KUKA KRL program: MyProgram_077().src

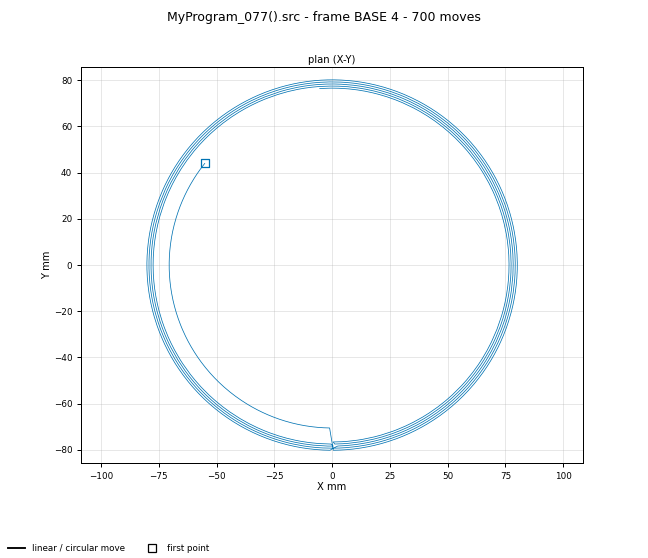
[picture p0: tool path of MyProgram_077().src in frame BASE 4, 700 of 700 moves have a stored position in this frame; points joined in program order, loops and branches not executed]
&ACCESS RVP
&REL 1
&PARAM TEMPLATE = C:\KRC\Roboter\Template\vorgabe
&PARAM EDITMASK = *
DEF MyProgram_077()
; ---- Setting reference (Base) ----
$BASE = BASE_DATA[4]

; --------------------------
; ---- Setting tool (TCP) ----
$TOOL = TOOL_DATA[3]
; --------------------------

$VEL.CP = VEL_APROX_PRINT
Startdeposition()
$VEL.CP = VEL_PRINT
LIN {X -55.1314,Y 43.9885,Z 79,A 136.1081,B 24.8816,C -2.5111,E1 24.8737,E2 308.1338} C_DIS
LIN {X -57.0335,Y 41.4919,Z 79,A 138.4284,B 24.8828,C -2.4992,E1 24.8699,E2 305.8307} C_DIS
LIN {X -58.5164,Y 39.3729,Z 79,A 140.5439,B 24.8833,C -2.4938,E1 24.8665,E2 303.7176} C_DIS
LIN {X -59.694,Y 37.5637,Z 79,A 142.4917,B 24.8833,C -2.4932,E1 24.8636,E2 301.7614} C_DIS
LIN {X -61.332,Y 34.8263,Z 79,A 145.2364,B 24.8837,C -2.4892,E1 24.8597,E2 299.012} C_DIS
LIN {X -62.6132,Y 32.4671,Z 79,A 147.3566,B 24.8844,C -2.4816,E1 24.857,E2 296.8988} C_DIS
LIN {X -63.7621,Y 30.1485,Z 79,A 149.3257,B 24.8853,C -2.4725,E1 24.8546,E2 294.9408} C_DIS
LIN {X -64.8254,Y 27.7886,Z 79,A 151.5952,B 24.8855,C -2.4698,E1 24.8521,E2 292.665} C_DIS
LIN {X -65.8013,Y 25.3913,Z 79,A 153.5568,B 24.8864,C -2.4604,E1 24.8501,E2 290.715} C_DIS
LIN {X -66.6884,Y 22.9605,Z 79,A 155.8268,B 24.8866,C -2.4576,E1 24.8479,E2 288.4387} C_DIS
LIN {X -67.5472,Y 20.2926,Z 79,A 158.0661,B 24.8874,C -2.4498,E1 24.8461,E2 286.2053} C_DIS
LIN {X -68.3657,Y 17.3357,Z 79,A 160.5177,B 24.8882,C -2.4412,E1 24.8443,E2 283.76} C_DIS
LIN {X -69.0025,Y 14.601,Z 79,A 162.777,B 24.8889,C -2.4335,E1 24.843,E2 281.5058} C_DIS
LIN {X -69.4922,Y 12.0572,Z 79,A 165.0492,B 24.8891,C -2.4305,E1 24.8418,E2 279.2273} C_DIS
LIN {X -69.9406,Y 9.0919,Z 79,A 167.3407,B 24.8901,C -2.4197,E1 24.8409,E2 276.948} C_DIS
LIN {X -70.2503,Y 6.2684,Z 79,A 169.5832,B 24.8909,C -2.4109,E1 24.8403,E2 274.7129} C_DIS
LIN {X -70.4338,Y 3.6722,Z 79,A 171.7072,B 24.8915,C -2.4044,E1 24.8399,E2 272.5917} C_DIS
LIN {X -70.5211,Y 1.0827,Z 79,A 174.0196,B 24.8917,C -2.4023,E1 24.8398,E2 270.2705} C_DIS
LIN {X -70.5092,Y -1.7264,Z 79,A 176.375,B 24.8922,C -2.3966,E1 24.8398,E2 267.9144} C_DIS
LIN {X -70.3982,Y -4.3149,Z 79,A 178.3488,B 24.8931,C -2.3871,E1 24.8402,E2 265.9514} C_DIS
LIN {X -70.1904,Y -6.9165,Z 79,A -179.3706,B 24.8934,C -2.384,E1 24.8408,E2 263.6647} C_DIS
LIN {X -69.8585,Y -9.7054,Z 79,A -177.1426,B 24.8941,C -2.3757,E1 24.8416,E2 261.4432} C_DIS
LIN {X -69.455,Y -12.2641,Z 79,A -175.0214,B 24.8946,C -2.3696,E1 24.8425,E2 259.324} C_DIS
LIN {X -68.8624,Y -15.2436,Z 79,A -172.5842,B 24.8954,C -2.3613,E1 24.8439,E2 256.8921} C_DIS
LIN {X -68.2017,Y -17.9741,Z 79,A -170.1696,B 24.8957,C -2.3573,E1 24.8456,E2 254.473} C_DIS
LIN {X -67.4309,Y -20.6756,Z 79,A -167.9357,B 24.8964,C -2.3495,E1 24.8474,E2 252.2449} C_DIS
LIN {X -66.6291,Y -23.1294,Z 79,A -165.8252,B 24.8969,C -2.3436,E1 24.8492,E2 250.1363} C_DIS
LIN {X -65.5843,Y -25.9438,Z 79,A -163.5524,B 24.8979,C -2.3329,E1 24.8515,E2 247.8763} C_DIS
LIN {X -64.775,Y -27.9042,Z 79,A -161.562,B 24.8978,C -2.334,E1 24.8537,E2 245.8724} C_DIS
LIN {X -63.4784,Y -30.7391,Z 79,A -159.2749,B 24.8989,C -2.3215,E1 24.8564,E2 243.6027} C_DIS
LIN {X -62.3075,Y -33.0479,Z 79,A -157.1577,B 24.8994,C -2.3161,E1 24.8591,E2 241.4871} C_DIS
LIN {X -61.053,Y -35.3117,Z 79,A -154.9151,B 24.8996,C -2.3136,E1 24.8622,E2 239.2385} C_DIS
LIN {X -59.5877,Y -37.7339,Z 79,A -152.4789,B 24.8998,C -2.3108,E1 24.8658,E2 236.7968} C_DIS
LIN {X -58.1586,Y -39.9012,Z 79,A -150.364,B 24.9003,C -2.3056,E1 24.8691,E2 234.6836} C_DIS
LIN {X -56.6707,Y -41.9875,Z 79,A -148.288,B 24.9007,C -2.3004,E1 24.8725,E2 232.61} C_DIS
LIN {X -54.7949,Y -44.4057,Z 79,A -145.763,B 24.9011,C -2.2955,E1 24.8769,E2 230.0849} C_DIS
LIN {X -52.7706,Y -46.7945,Z 79,A -143.2185,B 24.9016,C -2.2898,E1 24.8815,E2 227.5425} C_DIS
LIN {X -50.8754,Y -48.8473,Z 79,A -141.0304,B 24.9022,C -2.283,E1 24.8857,E2 225.3609} C_DIS
LIN {X -48.8605,Y -50.8627,Z 79,A -138.5931,B 24.9024,C -2.2811,E1 24.8906,E2 222.9182} C_DIS
LIN {X -46.6368,Y -52.9099,Z 79,A -136.1496,B 24.9028,C -2.276,E1 24.8956,E2 220.4769} C_DIS
LIN {X -44.1609,Y -54.9933,Z 79,A -133.5445,B 24.9033,C -2.2706,E1 24.9013,E2 217.8749} C_DIS
LIN {X -41.7925,Y -56.8134,Z 79,A -131.1597,B 24.9037,C -2.2654,E1 24.9066,E2 215.4938} C_DIS
LIN {X -39.3679,Y -58.5198,Z 79,A -128.7599,B 24.9041,C -2.2613,E1 24.9121,E2 213.0956} C_DIS
LIN {X -37.0061,Y -60.0423,Z 79,A -126.3522,B 24.9041,C -2.2608,E1 24.9178,E2 210.6814} C_DIS
LIN {X -34.7597,Y -61.3701,Z 79,A -124.3781,B 24.9047,C -2.2544,E1 24.9225,E2 208.7168} C_DIS
LIN {X -32.4884,Y -62.6022,Z 79,A -122.1216,B 24.9046,C -2.2555,E1 24.9281,E2 206.4514} C_DIS
LIN {X -30.1741,Y -63.7499,Z 79,A -120.1783,B 24.9051,C -2.2493,E1 24.933,E2 204.5179} C_DIS
LIN {X -27.8222,Y -64.8108,Z 79,A -117.9214,B 24.9049,C -2.2509,E1 24.9388,E2 202.2517} C_DIS
LIN {X -25.4477,Y -65.7792,Z 79,A -115.9713,B 24.9054,C -2.2457,E1 24.9438,E2 200.3098} C_DIS
LIN {X -22.9341,Y -66.6975,Z 79,A -113.6524,B 24.9052,C -2.2474,E1 24.95,E2 197.9823} C_DIS
LIN {X -20.263,Y -67.556,Z 79,A -111.4377,B 24.9055,C -2.2442,E1 24.9558,E2 195.7714} C_DIS
LIN {X -17.3572,Y -68.3602,Z 79,A -109.033,B 24.9057,C -2.2416,E1 24.9623,E2 193.3691} C_DIS
LIN {X -14.6256,Y -68.9972,Z 79,A -106.7919,B 24.9059,C -2.2396,E1 24.9684,E2 191.13} C_DIS
LIN {X -12.087,Y -69.4868,Z 79,A -104.5246,B 24.9056,C -2.2431,E1 24.9747,E2 188.8521} C_DIS
LIN {X -9.24,Y -69.9214,Z 79,A -102.2807,B 24.9059,C -2.2402,E1 24.9809,E2 186.6133} C_DIS
LIN {X -6.2929,Y -70.248,Z 79,A -100.0258,B 24.9062,C -2.2361,E1 24.9871,E2 184.3669} C_DIS
LIN {X -3.7214,Y -70.431,Z 79,A -97.9292,B 24.9062,C -2.2361,E1 24.993,E2 182.2693} C_DIS
LIN {X -1.0857,Y -70.521,Z 79,A -95.6624,B 24.9059,C -2.2397,E1 24.9993,E2 179.994} C_DIS
LIN {X -1.0857,Y -70.521,Z 79,A -95.6624,B 24.9059,C -2.2397,E1 24.9993,E2 179.994} C_DIS
Enddeposition()
LIN {X 0.5223,Y -80.1629,Z 80,A -94.9522,B 24.9201,C -2.0638,E1 25.0001,E2 179.7014} C_DIS
Startdeposition()
$VEL.CP = VEL_PRINT
LIN {X 3.5738,Y -80.0857,Z 80,A -91.9127,B 24.9181,C -2.0895,E1 25.0088,E2 176.6013} C_DIS
LIN {X 6.2912,Y -79.9181,Z 80,A -90.0185,B 24.9181,C -2.0889,E1 25.0141,E2 174.7096} C_DIS
LIN {X 9.0357,Y -79.6549,Z 80,A -87.8669,B 24.9177,C -2.0954,E1 25.0201,E2 172.544} C_DIS
LIN {X 12.4392,Y -79.1945,Z 80,A -85.4934,B 24.9177,C -2.0946,E1 25.0266,E2 170.1743} C_DIS
LIN {X 15.6125,Y -78.6306,Z 80,A -83.3311,B 24.9179,C -2.0923,E1 25.0325,E2 168.0202} C_DIS
LIN {X 18.3183,Y -78.0448,Z 80,A -81.1674,B 24.9173,C -2.0997,E1 25.0385,E2 165.8418} C_DIS
LIN {X 21.381,Y -77.2609,Z 80,A -79.2279,B 24.9179,C -2.0924,E1 25.0437,E2 163.9226} C_DIS
LIN {X 24.237,Y -76.415,Z 80,A -76.7008,B 24.9168,C -2.1069,E1 25.0505,E2 161.3657} C_DIS
LIN {X 27.8769,Y -75.1616,Z 80,A -74.34,B 24.9174,C -2.0985,E1 25.0566,E2 159.0296} C_DIS
LIN {X 30.4325,Y -74.1645,Z 80,A -72.076,B 24.9165,C -2.1105,E1 25.0626,E2 156.7422} C_DIS
LIN {X 33.383,Y -72.8834,Z 80,A -70.0419,B 24.9168,C -2.1058,E1 25.0677,E2 154.7241} C_DIS
LIN {X 36.0435,Y -71.606,Z 80,A -67.7149,B 24.916,C -2.1159,E1 25.0736,E2 152.3794} C_DIS
LIN {X 38.7509,Y -70.1782,Z 80,A -65.5829,B 24.9159,C -2.1179,E1 25.0788,E2 150.2488} C_DIS
LIN {X 41.2637,Y -68.7311,Z 80,A -63.4611,B 24.9155,C -2.1232,E1 25.0839,E2 148.121} C_DIS
LIN {X 43.8675,Y -67.0985,Z 80,A -61.3015,B 24.9152,C -2.1263,E1 25.089,E2 145.9611} C_DIS
LIN {X 46.5483,Y -65.2666,Z 80,A -59.038,B 24.915,C -2.1292,E1 25.0942,E2 143.6986} C_DIS
LIN {X 49.1868,Y -63.3027,Z 80,A -56.5823,B 24.9143,C -2.1374,E1 25.0997,E2 141.2324} C_DIS
LIN {X 51.8574,Y -61.1335,Z 80,A -54.1898,B 24.914,C -2.1408,E1 25.1048,E2 138.8411} C_DIS
LIN {X 54.4427,Y -58.8436,Z 80,A -51.7288,B 24.9136,C -2.1462,E1 25.1099,E2 136.3771} C_DIS
LIN {X 56.7655,Y -56.6064,Z 80,A -49.4236,B 24.9132,C -2.1518,E1 25.1145,E2 134.0685} C_DIS
LIN {X 58.9533,Y -54.3231,Z 80,A -47.1689,B 24.9127,C -2.1572,E1 25.1188,E2 131.8108} C_DIS
LIN {X 61.3516,Y -51.6011,Z 80,A -44.5862,B 24.9122,C -2.1635,E1 25.1235,E2 129.2249} C_DIS
LIN {X 63.3027,Y -49.1868,Z 80,A -42.3804,B 24.9118,C -2.1689,E1 25.1274,E2 127.0165} C_DIS
LIN {X 65.2666,Y -46.5483,Z 80,A -40.0511,B 24.9113,C -2.1746,E1 25.1312,E2 124.6851} C_DIS
LIN {X 67.0985,Y -43.8675,Z 80,A -37.7702,B 24.9109,C -2.1798,E1 25.1347,E2 122.4033} C_DIS
LIN {X 68.7749,Y -41.19,Z 80,A -35.5455,B 24.9104,C -2.1851,E1 25.138,E2 120.1774} C_DIS
LIN {X 70.2553,Y -38.6115,Z 80,A -33.4541,B 24.91,C -2.1902,E1 25.1408,E2 118.0849} C_DIS
LIN {X 71.6694,Y -35.9177,Z 80,A -31.2202,B 24.9093,C -2.1985,E1 25.1437,E2 115.8433} C_DIS
LIN {X 72.9727,Y -33.1892,Z 80,A -29.1799,B 24.9091,C -2.201,E1 25.1461,E2 113.8079} C_DIS
LIN {X 74.1645,Y -30.4325,Z 80,A -26.9676,B 24.9084,C -2.2096,E1 25.1485,E2 111.5875} C_DIS
LIN {X 75.3506,Y -27.3635,Z 80,A -24.62,B 24.9078,C -2.2167,E1 25.1508,E2 109.2362} C_DIS
LIN {X 76.4315,Y -24.1845,Z 80,A -22.1399,B 24.907,C -2.2267,E1 25.153,E2 106.7466} C_DIS
LIN {X 77.5189,Y -20.4316,Z 80,A -19.4725,B 24.9066,C -2.2314,E1 25.1549,E2 104.0834} C_DIS
LIN {X 78.2582,Y -17.3842,Z 80,A -17.344,B 24.9063,C -2.2348,E1 25.1563,E2 101.9592} C_DIS
LIN {X 78.8279,Y -14.5873,Z 80,A -15.2763,B 24.9057,C -2.2422,E1 25.1574,E2 99.8862} C_DIS
LIN {X 79.2987,Y -11.7628,Z 80,A -13.2188,B 24.9051,C -2.2491,E1 25.1583,E2 97.8246} C_DIS
LIN {X 79.6766,Y -8.836,Z 80,A -11.0985,B 24.9045,C -2.2562,E1 25.159,E2 95.7} C_DIS
LIN {X 79.9651,Y -5.6668,Z 80,A -8.7996,B 24.9038,C -2.2642,E1 25.1595,E2 93.3958} C_DIS
LIN {X 80.1418,Y -1.9398,Z 80,A -6.211,B 24.9033,C -2.2702,E1 25.1598,E2 90.8084} C_DIS
LIN {X 80.1574,Y 1.1669,Z 80,A -3.8994,B 24.9025,C -2.2802,E1 25.1598,E2 88.487} C_DIS
LIN {X 80.0402,Y 4.4763,Z 80,A -1.6758,B 24.9022,C -2.2831,E1 25.1594,E2 86.2697} C_DIS
LIN {X 79.8147,Y 7.4897,Z 80,A 0.4758,B 24.9016,C -2.2896,E1 25.1589,E2 84.1155} C_DIS
LIN {X 79.4367,Y 10.7888,Z 80,A 2.902,B 24.9009,C -2.2988,E1 25.1581,E2 81.682} C_DIS
LIN {X 78.9428,Y 13.9486,Z 80,A 5.1167,B 24.9004,C -2.3036,E1 25.1571,E2 79.4689} C_DIS
LIN {X 78.398,Y 16.7433,Z 80,A 7.168,B 24.8999,C -2.3104,E1 25.1559,E2 77.4136} C_DIS
LIN {X 77.6572,Y 19.8955,Z 80,A 9.4494,B 24.8993,C -2.3164,E1 25.1544,E2 75.1312} C_DIS
LIN {X 76.9876,Y 22.3515,Z 80,A 11.3758,B 24.8986,C -2.3252,E1 25.1529,E2 73.1948} C_DIS
LIN {X 75.804,Y 26.0855,Z 80,A 14.1035,B 24.898,C -2.3312,E1 25.1505,E2 70.4684} C_DIS
LIN {X 74.7866,Y 28.8732,Z 80,A 16.2095,B 24.8975,C -2.3369,E1 25.1484,E2 68.3608} C_DIS
LIN {X 73.5077,Y 31.9859,Z 80,A 18.5391,B 24.8971,C -2.3414,E1 25.1459,E2 66.0335} C_DIS
LIN {X 72.4161,Y 34.3876,Z 80,A 20.5035,B 24.8965,C -2.3491,E1 25.1436,E2 64.0613} C_DIS
LIN {X 70.8869,Y 37.437,Z 80,A 22.7713,B 24.8963,C -2.3504,E1 25.1407,E2 61.8024} C_DIS
LIN {X 69.5058,Y 39.9426,Z 80,A 24.807,B 24.8959,C -2.3556,E1 25.1379,E2 59.7651} C_DIS
LIN {X 67.9275,Y 42.5716,Z 80,A 27.0111,B 24.8953,C -2.3617,E1 25.1347,E2 57.5578} C_DIS
LIN {X 66.2424,Y 45.1494,Z 80,A 29.2856,B 24.8946,C -2.3696,E1 25.1311,E2 55.276} C_DIS
LIN {X 64.3571,Y 47.7997,Z 80,A 31.6145,B 24.8941,C -2.3754,E1 25.1273,E2 52.9446} C_DIS
LIN {X 62.2366,Y 50.528,Z 80,A 34.0403,B 24.8937,C -2.3799,E1 25.1231,E2 50.5195} C_DIS
LIN {X 60.0369,Y 53.1237,Z 80,A 36.4824,B 24.8932,C -2.3857,E1 25.1186,E2 48.0746} C_DIS
LIN {X 57.7753,Y 55.5742,Z 80,A 38.7345,B 24.8931,C -2.3868,E1 25.1143,E2 45.8297} C_DIS
LIN {X 55.4573,Y 57.8879,Z 80,A 41.1215,B 24.8925,C -2.3931,E1 25.1095,E2 43.4378} C_DIS
LIN {X 53.0243,Y 60.1252,Z 80,A 43.5607,B 24.8919,C -2.4002,E1 25.1045,E2 40.9917} C_DIS
LIN {X 50.4022,Y 62.3385,Z 80,A 45.8875,B 24.8919,C -2.4009,E1 25.0995,E2 38.672} C_DIS
LIN {X 47.7997,Y 64.3571,Z 80,A 48.2922,B 24.8913,C -2.4066,E1 25.0941,E2 36.2627} C_DIS
LIN {X 45.1494,Y 66.2424,Z 80,A 50.5578,B 24.8911,C -2.4086,E1 25.0889,E2 33.9999} C_DIS
LIN {X 42.5716,Y 67.9275,Z 80,A 52.7489,B 24.8908,C -2.4117,E1 25.0838,E2 31.8086} C_DIS
LIN {X 39.9426,Y 69.5058,Z 80,A 54.8968,B 24.8907,C -2.4136,E1 25.0786,E2 29.6629} C_DIS
LIN {X 37.437,Y 70.8869,Z 80,A 57.0166,B 24.8902,C -2.4186,E1 25.0734,E2 27.5373} C_DIS
LIN {X 34.3002,Y 72.4573,Z 80,A 59.5962,B 24.8897,C -2.4238,E1 25.0669,E2 24.9523} C_DIS
LIN {X 31.0661,Y 73.9011,Z 80,A 62.0481,B 24.8897,C -2.4241,E1 25.0606,E2 22.5054} C_DIS
LIN {X 28.2922,Y 75.0069,Z 80,A 64.1764,B 24.8895,C -2.426,E1 25.0551,E2 20.3772} C_DIS
LIN {X 25.5016,Y 76.001,Z 80,A 66.2855,B 24.8895,C -2.4276,E1 25.0495,E2 18.2686} C_DIS
LIN {X 22.3279,Y 76.9943,Z 80,A 68.7742,B 24.8889,C -2.4326,E1 25.0428,E2 15.7724} C_DIS
LIN {X 18.9606,Y 77.8907,Z 80,A 71.1195,B 24.8892,C -2.4298,E1 25.0365,E2 13.4372} C_DIS
LIN {X 16.0165,Y 78.5487,Z 80,A 73.323,B 24.889,C -2.4322,E1 25.0305,E2 11.2309} C_DIS
LIN {X 12.7079,Y 79.153,Z 80,A 75.6013,B 24.8892,C -2.4294,E1 25.0242,E2 8.9617} C_DIS
LIN {X 9.9558,Y 79.5454,Z 80,A 77.6865,B 24.8889,C -2.4327,E1 25.0184,E2 6.8704} C_DIS
LIN {X 6.8781,Y 79.8707,Z 80,A 79.89,B 24.8889,C -2.4327,E1 25.0123,E2 4.6683} C_DIS
LIN {X 3.8564,Y 80.0735,Z 80,A 82.0431,B 24.8889,C -2.4323,E1 25.0063,E2 2.5169} C_DIS
LIN {X 0.8877,Y 80.1613,Z 80,A 84.1718,B 24.8889,C -2.4322,E1 25.0004,E2 0.3887} C_DIS
LIN {X -1.9949,Y 80.1403,Z 80,A 86.2199,B 24.8891,C -2.4314,E1 24.9947,E2 -1.6575} C_DIS
LIN {X -4.9158,Y 80.0145,Z 80,A 88.2536,B 24.8893,C -2.429,E1 24.989,E2 -3.6862} C_DIS
LIN {X -7.4897,Y 79.8147,Z 80,A 90.1437,B 24.8893,C -2.4294,E1 24.9838,E2 -5.5782} C_DIS
LIN {X -10.7888,Y 79.4367,Z 80,A 92.5901,B 24.8892,C -2.4301,E1 24.977,E2 -8.0278} C_DIS
LIN {X -13.9486,Y 78.9428,Z 80,A 94.871,B 24.8893,C -2.4283,E1 24.9707,E2 -10.3067} C_DIS
LIN {X -16.7433,Y 78.398,Z 80,A 96.9202,B 24.8895,C -2.427,E1 24.9651,E2 -12.3552} C_DIS
LIN {X -19.8955,Y 77.6572,Z 80,A 99.1945,B 24.8898,C -2.4237,E1 24.9589,E2 -14.6248} C_DIS
LIN {X -22.3544,Y 76.9868,Z 80,A 101.1478,B 24.8896,C -2.4254,E1 24.9537,E2 -16.5853} C_DIS
LIN {X -26.0855,Y 75.804,Z 80,A 103.8912,B 24.89,C -2.4206,E1 24.9464,E2 -19.3223} C_DIS
LIN {X -28.8732,Y 74.7866,Z 80,A 106.017,B 24.8903,C -2.4179,E1 24.9409,E2 -21.4463} C_DIS
LIN {X -31.9858,Y 73.5077,Z 80,A 108.3575,B 24.8907,C -2.4128,E1 24.9349,E2 -23.7799} C_DIS
LIN {X -34.3876,Y 72.4161,Z 80,A 110.3522,B 24.8907,C -2.4128,E1 24.9298,E2 -25.7798} C_DIS
LIN {X -37.437,Y 70.8869,Z 80,A 112.6419,B 24.8915,C -2.4049,E1 24.9242,E2 -28.0567} C_DIS
LIN {X -39.9426,Y 69.5058,Z 80,A 114.6975,B 24.8918,C -2.4016,E1 24.9192,E2 -30.1106} C_DIS
LIN {X -42.5716,Y 67.9275,Z 80,A 116.9235,B 24.892,C -2.3986,E1 24.9139,E2 -32.3362} C_DIS
LIN {X -45.1494,Y 66.2424,Z 80,A 119.2205,B 24.8922,C -2.3969,E1 24.9085,E2 -34.6368} C_DIS
LIN {X -47.7997,Y 64.3571,Z 80,A 121.5729,B 24.8926,C -2.3929,E1 24.9032,E2 -36.9879} C_DIS
LIN {X -50.528,Y 62.2366,Z 80,A 124.0229,B 24.8931,C -2.3871,E1 24.8979,E2 -39.4333} C_DIS
LIN {X -53.1237,Y 60.0369,Z 80,A 126.4897,B 24.8935,C -2.3826,E1 24.8927,E2 -41.8989} C_DIS
LIN {X -55.5742,Y 57.7753,Z 80,A 128.7644,B 24.8942,C -2.3742,E1 24.8881,E2 -44.163} C_DIS
LIN {X -57.8879,Y 55.4573,Z 80,A 131.1754,B 24.8946,C -2.3704,E1 24.8833,E2 -46.5753} C_DIS
LIN {X -60.1252,Y 53.0243,Z 80,A 133.6393,B 24.8949,C -2.3672,E1 24.8787,E2 -49.0424} C_DIS
LIN {X -62.3385,Y 50.4022,Z 80,A 135.9889,B 24.8957,C -2.3582,E1 24.8746,E2 -51.3814} C_DIS
LIN {X -64.3571,Y 47.7997,Z 80,A 138.4176,B 24.896,C -2.3538,E1 24.8705,E2 -53.8114} C_DIS
LIN {X -66.2424,Y 45.1494,Z 80,A 140.7052,B 24.8967,C -2.3466,E1 24.8668,E2 -56.0929} C_DIS
LIN {X -67.9275,Y 42.5716,Z 80,A 142.931,B 24.8972,C -2.3411,E1 24.8635,E2 -58.3168} C_DIS
LIN {X -69.5058,Y 39.9426,Z 80,A 145.086,B 24.8978,C -2.3339,E1 24.8605,E2 -60.4659} C_DIS
LIN {X -70.8869,Y 37.437,Z 80,A 147.2257,B 24.8981,C -2.3304,E1 24.8576,E2 -62.6086} C_DIS
LIN {X -72.4161,Y 34.3876,Z 80,A 149.5869,B 24.8989,C -2.3213,E1 24.8547,E2 -64.9607} C_DIS
LIN {X -73.5077,Y 31.9859,Z 80,A 151.584,B 24.8991,C -2.3185,E1 24.8525,E2 -66.9621} C_DIS
LIN {X -74.7948,Y 28.8515,Z 80,A 154.0385,B 24.8997,C -2.312,E1 24.8499,E2 -69.4148} C_DIS
LIN {X -75.9027,Y 25.7931,Z 80,A 156.3282,B 24.9004,C -2.304,E1 24.8478,E2 -71.6984} C_DIS
LIN {X -76.9943,Y 22.3279,Z 80,A 159.0891,B 24.9007,C -2.3001,E1 24.8456,E2 -74.466} C_DIS
LIN {X -77.8907,Y 18.9606,Z 80,A 161.4535,B 24.9017,C -2.2891,E1 24.844,E2 -76.8179} C_DIS
LIN {X -78.5198,Y 16.1591,Z 80,A 163.4998,B 24.9023,C -2.2825,E1 24.8428,E2 -78.8604} C_DIS
LIN {X -79.0431,Y 13.3669,Z 80,A 165.555,B 24.9028,C -2.2767,E1 24.8418,E2 -80.914} C_DIS
LIN {X -79.4633,Y 10.5895,Z 80,A 167.6778,B 24.9031,C -2.2733,E1 24.841,E2 -83.0413} C_DIS
LIN {X -79.8411,Y 7.2032,Z 80,A 170.0244,B 24.9039,C -2.2632,E1 24.8403,E2 -85.378} C_DIS
LIN {X -80.0708,Y 3.9061,Z 80,A 172.4309,B 24.9044,C -2.2568,E1 24.8399,E2 -87.7836} C_DIS
LIN {X -80.1613,Y 0.8877,Z 80,A 174.553,B 24.9051,C -2.249,E1 24.8398,E2 -89.8999} C_DIS
LIN {X -80.1403,Y -1.9949,Z 80,A 176.715,B 24.9054,C -2.2451,E1 24.8398,E2 -92.0656} C_DIS
LIN {X -79.9844,Y -5.3822,Z 80,A 179.0573,B 24.9063,C -2.2354,E1 24.8402,E2 -94.3987} C_DIS
LIN {X -79.7234,Y -8.4054,Z 80,A -178.7025,B 24.9067,C -2.2304,E1 24.8408,E2 -96.6404} C_DIS
LIN {X -79.3345,Y -11.5134,Z 80,A -176.592,B 24.9075,C -2.2201,E1 24.8416,E2 -98.7389} C_DIS
LIN {X -78.9428,Y -13.9486,Z 80,A -174.6334,B 24.9075,C -2.2197,E1 24.8426,E2 -100.7082} C_DIS
LIN {X -78.398,Y -16.7433,Z 80,A -172.6016,B 24.9081,C -2.2133,E1 24.8437,E2 -102.7368} C_DIS
LIN {X -77.6572,Y -19.8955,Z 80,A -170.2891,B 24.9087,C -2.2063,E1 24.8452,E2 -105.046} C_DIS
LIN {X -76.9868,Y -22.3544,Z 80,A -168.3273,B 24.9088,C -2.2044,E1 24.8467,E2 -107.0147} C_DIS
LIN {X -75.804,Y -26.0855,Z 80,A -165.573,B 24.9096,C -2.195,E1 24.8492,E2 -109.7623} C_DIS
LIN {X -74.7866,Y -28.8732,Z 80,A -163.4397,B 24.9101,C -2.1892,E1 24.8513,E2 -111.8937} C_DIS
LIN {X -73.5077,Y -31.9858,Z 80,A -161.0918,B 24.9108,C -2.1809,E1 24.8538,E2 -114.2349} C_DIS
LIN {X -72.4161,Y -34.3876,Z 80,A -159.0914,B 24.911,C -2.1786,E1 24.8562,E2 -116.2406} C_DIS
LIN {X -70.8869,Y -37.437,Z 80,A -156.7961,B 24.9118,C -2.1682,E1 24.8591,E2 -118.5235} C_DIS
LIN {X -69.5058,Y -39.9426,Z 80,A -154.7361,B 24.9122,C -2.1632,E1 24.8619,E2 -120.5822} C_DIS
LIN {X -67.9275,Y -42.5716,Z 80,A -152.5063,B 24.9126,C -2.1585,E1 24.8652,E2 -122.8122} C_DIS
LIN {X -66.2424,Y -45.1494,Z 80,A -150.2062,B 24.9129,C -2.1555,E1 24.8687,E2 -125.1168} C_DIS
LIN {X -64.3571,Y -47.7997,Z 80,A -147.8518,B 24.9132,C -2.1506,E1 24.8726,E2 -127.4709} C_DIS
LIN {X -62.2366,Y -50.528,Z 80,A -145.4006,B 24.9138,C -2.1444,E1 24.8769,E2 -129.9187} C_DIS
LIN {X -60.0552,Y -53.1031,Z 80,A -142.9422,B 24.9141,C -2.1401,E1 24.8814,E2 -132.3782} C_DIS
LIN {X -57.7753,Y -55.5742,Z 80,A -140.6598,B 24.9148,C -2.1317,E1 24.8857,E2 -134.6504} C_DIS
LIN {X -55.4573,Y -57.8879,Z 80,A -138.2506,B 24.915,C -2.1287,E1 24.8905,E2 -137.0625} C_DIS
LIN {X -53.0243,Y -60.1252,Z 80,A -135.7897,B 24.9152,C -2.1267,E1 24.8957,E2 -139.5285} C_DIS
LIN {X -50.2555,Y -62.4575,Z 80,A -133.2988,B 24.9158,C -2.1193,E1 24.901,E2 -142.0114} C_DIS
LIN {X -47.755,Y -64.3902,Z 80,A -131.0018,B 24.916,C -2.1164,E1 24.9061,E2 -144.3096} C_DIS
LIN {X -45.1494,Y -66.2424,Z 80,A -128.7381,B 24.9163,C -2.1121,E1 24.9113,E2 -146.5709} C_DIS
LIN {X -42.5716,Y -67.9275,Z 80,A -126.5186,B 24.9166,C -2.1093,E1 24.9165,E2 -148.7907} C_DIS
LIN {X -39.9426,Y -69.5058,Z 80,A -124.3705,B 24.9169,C -2.105,E1 24.9217,E2 -150.9351} C_DIS
LIN {X -37.437,Y -70.8869,Z 80,A -122.2381,B 24.9169,C -2.1047,E1 24.9269,E2 -153.0728} C_DIS
LIN {X -34.3876,Y -72.4161,Z 80,A -119.7738,B 24.9171,C -2.1025,E1 24.9331,E2 -155.5384} C_DIS
LIN {X -31.3542,Y -73.7797,Z 80,A -117.3961,B 24.9173,C -2.1,E1 24.9392,E2 -157.9157} C_DIS
LIN {X -28.2922,Y -75.0069,Z 80,A -115.0438,B 24.9175,C -2.0977,E1 24.9453,E2 -160.2674} C_DIS
LIN {X -25.5016,Y -76.001,Z 80,A -112.9269,B 24.9176,C -2.0959,E1 24.9509,E2 -162.3843} C_DIS
LIN {X -22.3279,Y -76.9943,Z 80,A -110.4304,B 24.9175,C -2.0977,E1 24.9576,E2 -164.8891} C_DIS
LIN {X -18.9281,Y -77.8985,Z 80,A -108.0705,B 24.9179,C -2.0918,E1 24.964,E2 -167.2386} C_DIS
LIN {X -16.1591,Y -78.5198,Z 80,A -106.0453,B 24.918,C -2.0909,E1 24.9695,E2 -169.2639} C_DIS
LIN {X -13.3669,Y -79.0431,Z 80,A -104.003,B 24.918,C -2.0905,E1 24.9751,E2 -171.3075} C_DIS
LIN {X -10.5895,Y -79.4633,Z 80,A -101.8943,B 24.9178,C -2.093,E1 24.981,E2 -173.4237} C_DIS
LIN {X -7.2032,Y -79.8411,Z 80,A -99.5638,B 24.9181,C -2.0898,E1 24.9874,E2 -175.7478} C_DIS
LIN {X -3.9061,Y -80.0708,Z 80,A -97.1746,B 24.9181,C -2.0906,E1 24.9941,E2 -178.1398} C_DIS
LIN {X -0.8877,Y -80.1613,Z 80,A -95.0179,B 24.9181,C -2.0909,E1 25.0001,E2 -180.2975} C_DIS
LIN {X -0.8877,Y -80.1613,Z 80,A -95.0179,B 24.9181,C -2.0909,E1 25.0001,E2 -180.2975} C_DIS
Enddeposition()
LIN {X 0.5113,Y -79.2679,Z 80,A -94.2684,B 24.9173,C -2.0993,E1 25.0023,E2 -181.0667} C_DIS
Startdeposition()
$VEL.CP = VEL_PRINT
LIN {X -4.0138,Y -79.1697,Z 80,A -98.6051,B 24.9198,C -2.0683,E1 24.99,E2 -176.656} C_DIS
LIN {X -6.7676,Y -78.9826,Z 80,A -100.4551,B 24.9195,C -2.0724,E1 24.9849,E2 -174.8149} C_DIS
LIN {X -10.0746,Y -78.6285,Z 80,A -102.8222,B 24.9193,C -2.0738,E1 24.9783,E2 -172.4496} C_DIS
LIN {X -12.5662,Y -78.2702,Z 80,A -105.5536,B 24.9213,C -2.0491,E1 24.9706,E2 -169.6568} C_DIS
LIN {X -16.8137,Y -77.4676,Z 80,A -107.3755,B 24.9184,C -2.0864,E1 24.9659,E2 -167.9215} C_DIS
LIN {X -18.8261,Y -77.0033,Z 80,A -109.0895,B 24.9188,C -2.081,E1 24.9611,E2 -166.1924} C_DIS
LIN {X -21.2667,Y -76.3647,Z 80,A -110.994,B 24.9188,C -2.0799,E1 24.956,E2 -164.2822} C_DIS
LIN {X -24.2861,Y -75.4594,Z 80,A -113.3546,B 24.9189,C -2.0792,E1 24.9497,E2 -161.9161} C_DIS
LIN {X -27.2132,Y -74.4538,Z 80,A -115.6394,B 24.9189,C -2.0798,E1 24.9437,E2 -159.6282} C_DIS
LIN {X -30.2979,Y -73.2522,Z 80,A -118.2875,B 24.9192,C -2.0753,E1 24.9368,E2 -156.9633} C_DIS
LIN {X -33.4153,Y -71.8841,Z 80,A -121.0471,B 24.9196,C -2.07,E1 24.9297,E2 -154.1844} C_DIS
LIN {X -36.457,Y -70.3911,Z 80,A -123.6261,B 24.9196,C -2.0696,E1 24.9233,E2 -151.5974} C_DIS
LIN {X -39.7085,Y -68.6092,Z 80,A -125.5055,B 24.9177,C -2.0946,E1 24.9189,E2 -149.772} C_DIS
LIN {X -42.3138,Y -67.0343,Z 80,A -127.8259,B 24.9177,C -2.0946,E1 24.9133,E2 -147.4444} C_DIS
LIN {X -44.2626,Y -65.7631,Z 80,A -129.4834,B 24.9175,C -2.098,E1 24.9095,E2 -145.7893} C_DIS
LIN {X -46.8663,Y -63.9333,Z 80,A -131.8488,B 24.9173,C -2.1001,E1 24.9041,E2 -143.4207} C_DIS
LIN {X -49.9257,Y -61.5739,Z 80,A -134.5716,B 24.9167,C -2.1069,E1 24.8982,E2 -140.7042} C_DIS
LIN {X -52.3242,Y -59.5496,Z 80,A -136.9255,B 24.9166,C -2.109,E1 24.8932,E2 -138.3461} C_DIS
LIN {X -54.7702,Y -57.308,Z 80,A -139.3014,B 24.9162,C -2.1144,E1 24.8883,E2 -135.9733} C_DIS
LIN {X -57.1732,Y -54.9105,Z 80,A -141.5179,B 24.9153,C -2.1257,E1 24.884,E2 -133.7744} C_DIS
LIN {X -58.8911,Y -53.0644,Z 80,A -143.2954,B 24.9148,C -2.1309,E1 24.8807,E2 -132.0013} C_DIS
LIN {X -60.6587,Y -51.0358,Z 80,A -145.6034,B 24.9152,C -2.1259,E1 24.8764,E2 -129.6709} C_DIS
LIN {X -62.7691,Y -48.4145,Z 80,A -147.9945,B 24.9147,C -2.1327,E1 24.8723,E2 -127.2849} C_DIS
LIN {X -64.6887,Y -45.8189,Z 80,A -150.5532,B 24.9147,C -2.1327,E1 24.8681,E2 -124.7136} C_DIS
LIN {X -66.3758,Y -43.3389,Z 80,A -152.5367,B 24.9139,C -2.1429,E1 24.8651,E2 -122.7444} C_DIS
LIN {X -68.1145,Y -40.551,Z 80,A -154.8902,B 24.9133,C -2.1496,E1 24.8616,E2 -120.3949} C_DIS
LIN {X -70.122,Y -36.9703,Z 80,A -157.8284,B 24.9126,C -2.1583,E1 24.8577,E2 -117.4619} C_DIS
LIN {X -71.5661,Y -34.0924,Z 80,A -160.2828,B 24.9124,C -2.1615,E1 24.8547,E2 -115.0019} C_DIS
LIN {X -72.9902,Y -30.9254,Z 80,A -162.811,B 24.9118,C -2.1681,E1 24.8519,E2 -112.4757} C_DIS
LIN {X -74.0318,Y -28.3422,Z 80,A -165.0102,B 24.9118,C -2.1693,E1 24.8496,E2 -110.2669} C_DIS
LIN {X -75.3019,Y -24.7686,Z 80,A -167.5009,B 24.9106,C -2.1836,E1 24.8474,E2 -107.7961} C_DIS
LIN {X -76.3594,Y -21.2859,Z 80,A -169.7674,B 24.9092,C -2.2006,E1 24.8456,E2 -105.5572} C_DIS
LIN {X -76.8904,Y -19.2802,Z 80,A -171.6426,B 24.9096,C -2.1957,E1 24.8443,E2 -103.6594} C_DIS
LIN {X -77.5028,Y -16.6522,Z 80,A -173.7398,B 24.9094,C -2.198,E1 24.843,E2 -101.5554} C_DIS
LIN {X -78.1257,Y -13.4323,Z 80,A -176.0063,B 24.9086,C -2.2079,E1 24.8419,E2 -99.299} C_DIS
LIN {X -78.5695,Y -10.5277,Z 80,A -178.1071,B 24.908,C -2.2151,E1 24.841,E2 -97.2029} C_DIS
LIN {X -78.9134,Y -7.5202,Z 80,A 179.6358,B 24.9075,C -2.2203,E1 24.8404,E2 -94.9446} C_DIS
LIN {X -79.1567,Y -4.2565,Z 80,A 177.3321,B 24.9068,C -2.2293,E1 24.84,E2 -92.6485} C_DIS
LIN {X -79.2596,Y -1.3587,Z 80,A 175.0556,B 24.9066,C -2.2314,E1 24.8398,E2 -90.3636} C_DIS
LIN {X -79.2474,Y 1.9404,Z 80,A 172.8177,B 24.9056,C -2.2427,E1 24.8398,E2 -88.139} C_DIS
LIN {X -79.134,Y 4.672,Z 80,A 170.6618,B 24.9055,C -2.2445,E1 24.8402,E2 -85.9745} C_DIS
LIN {X -78.8805,Y 7.8586,Z 80,A 168.3804,B 24.9048,C -2.2526,E1 24.8407,E2 -83.6986} C_DIS
LIN {X -78.4945,Y 11.07,Z 80,A 166.07,B 24.9041,C -2.2607,E1 24.8416,E2 -81.3938} C_DIS
LIN {X -77.9894,Y 14.1988,Z 80,A 163.7311,B 24.9036,C -2.2668,E1 24.8427,E2 -79.0555} C_DIS
LIN {X -77.3665,Y 17.2752,Z 80,A 161.4663,B 24.903,C -2.274,E1 24.844,E2 -76.7946} C_DIS
LIN {X -76.5566,Y 20.5675,Z 80,A 159.1924,B 24.902,C -2.286,E1 24.8455,E2 -74.5362} C_DIS
LIN {X -75.9121,Y 22.8311,Z 80,A 157.257,B 24.902,C -2.2855,E1 24.8471,E2 -72.5885} C_DIS
LIN {X -74.6797,Y 26.5857,Z 80,A 154.4529,B 24.9011,C -2.2956,E1 24.8496,E2 -69.7924} C_DIS
LIN {X -72.1837,Y 32.764,Z 80,A 149.4813,B 24.9002,C -2.3063,E1 24.8549,E2 -64.8186} C_DIS
LIN {X -70.8396,Y 35.5777,Z 80,A 146.8867,B 24.9004,C -2.3044,E1 24.8581,E2 -62.2057} C_DIS
LIN {X -68.8857,Y 39.2273,Z 80,A 144.2117,B 24.8989,C -2.3209,E1 24.8617,E2 -59.556} C_DIS
LIN {X -67.1404,Y 42.1441,Z 80,A 141.7327,B 24.8984,C -2.3273,E1 24.8653,E2 -57.0794} C_DIS
LIN {X -65.2345,Y 45.0383,Z 80,A 139.2609,B 24.8977,C -2.335,E1 24.8692,E2 -54.6138} C_DIS
LIN {X -62.6904,Y 48.5166,Z 80,A 136.2649,B 24.8967,C -2.3463,E1 24.8742,E2 -51.6303} C_DIS
LIN {X -61.3561,Y 50.1938,Z 80,A 134.5623,B 24.8967,C -2.3464,E1 24.8772,E2 -49.9201} C_DIS
LIN {X -59.275,Y 52.6351,Z 80,A 132.2252,B 24.8962,C -2.3518,E1 24.8814,E2 -47.5853} C_DIS
LIN {X -56.8434,Y 55.2527,Z 80,A 129.5953,B 24.8958,C -2.3569,E1 24.8865,E2 -44.9561} C_DIS
LIN {X -54.8409,Y 57.2403,Z 80,A 127.6328,B 24.8952,C -2.3637,E1 24.8904,E2 -43.0015} C_DIS
LIN {X -52.5304,Y 59.3681,Z 80,A 125.2586,B 24.8949,C -2.3662,E1 24.8953,E2 -40.6239} C_DIS
LIN {X -50.0292,Y 61.4901,Z 80,A 122.9397,B 24.8944,C -2.3727,E1 24.9003,E2 -38.3117} C_DIS
LIN {X -47.3867,Y 63.5492,Z 80,A 120.5322,B 24.8939,C -2.3781,E1 24.9056,E2 -35.9083} C_DIS
LIN {X -45.4927,Y 64.9185,Z 80,A 118.7987,B 24.8937,C -2.3803,E1 24.9096,E2 -34.1741} C_DIS
LIN {X -42.7261,Y 66.7714,Z 80,A 116.4668,B 24.8931,C -2.3869,E1 24.915,E2 -31.8501} C_DIS
LIN {X -39.9885,Y 68.4471,Z 80,A 114.0141,B 24.8931,C -2.3876,E1 24.9209,E2 -29.3916} C_DIS
LIN {X -37.0315,Y 70.0899,Z 80,A 111.6242,B 24.8925,C -2.3932,E1 24.9267,E2 -27.0083} C_DIS
LIN {X -34.9896,Y 71.1307,Z 80,A 109.8217,B 24.8926,C -2.392,E1 24.9313,E2 -25.1982} C_DIS
LIN {X -31.2941,Y 72.8321,Z 80,A 106.6636,B 24.8928,C -2.3906,E1 24.9394,E2 -22.0292} C_DIS
LIN {X -27.32,Y 74.4148,Z 80,A 103.5265,B 24.8925,C -2.3935,E1 24.9475,E2 -18.8924} C_DIS
LIN {X -23.9263,Y 75.5755,Z 80,A 101.2373,B 24.8915,C -2.4045,E1 24.9536,E2 -16.6253} C_DIS
LIN {X -20.7568,Y 76.5055,Z 80,A 98.8568,B 24.8913,C -2.4072,E1 24.96,E2 -14.2474} C_DIS
LIN {X -17.777,Y 77.2522,Z 80,A 96.5978,B 24.8912,C -2.4082,E1 24.9661,E2 -11.9878} C_DIS
LIN {X -15.2631,Y 77.7884,Z 80,A 94.8012,B 24.8909,C -2.4114,E1 24.971,E2 -10.1966} C_DIS
LIN {X -12.0464,Y 78.3506,Z 80,A 92.397,B 24.8909,C -2.4119,E1 24.9776,E2 -7.7914} C_DIS
LIN {X -8.6299,Y 78.7997,Z 80,A 89.9121,B 24.8907,C -2.4135,E1 24.9845,E2 -5.3086} C_DIS
LIN {X -5.1887,Y 79.1009,Z 80,A 86.6523,B 24.8925,C -2.3938,E1 24.9937,E2 -2.0008} C_DIS
LIN {X -1.2117,Y 79.2623,Z 80,A 83.5052,B 24.8931,C -2.3871,E1 25.0025,E2 1.1623} C_DIS
LIN {X 3.5216,Y 79.193,Z 80,A 81.4591,B 24.8896,C -2.4253,E1 25.008,E2 3.1173} C_DIS
LIN {X 5.8486,Y 79.0548,Z 80,A 78.7842,B 24.8921,C -2.3978,E1 25.0156,E2 5.8563} C_DIS
LIN {X 9.4381,Y 78.707,Z 80,A 76.1148,B 24.8923,C -2.3956,E1 25.023,E2 8.529} C_DIS
LIN {X 13.211,Y 78.1627,Z 80,A 74.1878,B 24.8903,C -2.4179,E1 25.0282,E2 10.4011} C_DIS
LIN {X 15.9593,Y 77.648,Z 80,A 72.146,B 24.8904,C -2.4164,E1 25.0338,E2 12.4439} C_DIS
LIN {X 19.2266,Y 76.9039,Z 80,A 69.6599,B 24.8907,C -2.4133,E1 25.0406,E2 14.9339} C_DIS
LIN {X 22.4853,Y 76.0154,Z 80,A 67.2096,B 24.8909,C -2.4114,E1 25.0471,E2 17.3846} C_DIS
LIN {X 25.5399,Y 75.0445,Z 80,A 64.9222,B 24.8909,C -2.4103,E1 25.0532,E2 19.6702} C_DIS
LIN {X 29.3063,Y 73.6556,Z 80,A 62.0878,B 24.891,C -2.4095,E1 25.0606,E2 22.5004} C_DIS
LIN {X 32.0791,Y 72.491,Z 80,A 59.7827,B 24.8916,C -2.4034,E1 25.0665,E2 24.8146} C_DIS
LIN {X 37.3364,Y 69.9289,Z 80,A 55.5971,B 24.892,C -2.3993,E1 25.077,E2 28.9984} C_DIS
LIN {X 40.2878,Y 68.2702,Z 80,A 53.2269,B 24.892,C -2.3981,E1 25.0827,E2 31.3643} C_DIS
LIN {X 42.9021,Y 66.6584,Z 80,A 50.9443,B 24.8925,C -2.3929,E1 25.0881,E2 33.652} C_DIS
LIN {X 45.7454,Y 64.7409,Z 80,A 48.4094,B 24.8931,C -2.3871,E1 25.0939,E2 36.1919} C_DIS
LIN {X 49.7752,Y 61.6959,Z 80,A 45.2708,B 24.8923,C -2.3959,E1 25.1008,E2 39.2982} C_DIS
LIN {X 51.3615,Y 60.3815,Z 80,A 43.3882,B 24.8936,C -2.3813,E1 25.1049,E2 41.2082} C_DIS
LIN {X 53.8413,Y 58.1821,Z 80,A 40.9062,B 24.8942,C -2.374,E1 25.1101,E2 43.6976} C_DIS
LIN {X 55.6548,Y 56.4489,Z 80,A 38.6665,B 24.8957,C -2.3574,E1 25.1146,E2 45.967} C_DIS
LIN {X 57.8916,Y 54.1528,Z 80,A 36.414,B 24.896,C -2.3543,E1 25.1189,E2 48.2171} C_DIS
LIN {X 60.5042,Y 51.2174,Z 80,A 34.2634,B 24.8947,C -2.3687,E1 25.1227,E2 50.324} C_DIS
LIN {X 62.2794,Y 49.043,Z 80,A 32.0333,B 24.8957,C -2.3578,E1 25.1267,E2 52.5694} C_DIS
LIN {X 65.0268,Y 45.3371,Z 80,A 29.0227,B 24.8955,C -2.3595,E1 25.1316,E2 55.5614} C_DIS
LIN {X 66.3816,Y 43.33,Z 80,A 26.9726,B 24.8967,C -2.3458,E1 25.1348,E2 57.6336} C_DIS
LIN {X 68.1089,Y 40.5605,Z 80,A 24.4993,B 24.8976,C -2.3362,E1 25.1384,E2 60.1171} C_DIS
LIN {X 69.9158,Y 37.3607,Z 80,A 21.9773,B 24.8979,C -2.3331,E1 25.1418,E2 62.6331} C_DIS
LIN {X 71.9242,Y 33.3282,Z 80,A 19.0734,B 24.8977,C -2.335,E1 25.1453,E2 65.5169} C_DIS
LIN {X 72.9491,Y 31.0225,Z 80,A 16.9121,B 24.8991,C -2.3194,E1 25.1477,E2 67.7034} C_DIS
LIN {X 74.7297,Y 26.4464,Z 80,A 13.5313,B 24.8995,C -2.3143,E1 25.1511,E2 71.0773} C_DIS
LIN {X 75.6779,Y 23.5965,Z 80,A 11.2646,B 24.9003,C -2.3049,E1 25.153,E2 73.3535} C_DIS
LIN {X 76.6161,Y 20.3474,Z 80,A 8.7763,B 24.9011,C -2.2961,E1 25.1549,E2 75.8482} C_DIS
LIN {X 77.4058,Y 17.0971,Z 80,A 6.5358,B 24.9012,C -2.2943,E1 25.1563,E2 78.0799} C_DIS
LIN {X 77.9682,Y 14.3165,Z 80,A 3.9669,B 24.9032,C -2.2718,E1 25.1577,E2 80.687} C_DIS
LIN {X 78.5057,Y 10.9913,Z 80,A 1.0713,B 24.905,C -2.2499,E1 25.1588,E2 83.6173} C_DIS
LIN {X 78.9907,Y 6.6682,Z 80,A -0.8872,B 24.9027,C -2.2769,E1 25.1593,E2 85.5003} C_DIS
LIN {X 79.1484,Y 4.4108,Z 80,A -2.747,B 24.9038,C -2.2647,E1 25.1596,E2 87.3779} C_DIS
LIN {X 79.2647,Y 1.0603,Z 80,A -5.2069,B 24.9045,C -2.2558,E1 25.1598,E2 89.8442} C_DIS
LIN {X 79.1987,Y -3.3892,Z 80,A -8.2981,B 24.9051,C -2.2495,E1 25.1596,E2 92.9319} C_DIS
LIN {X 78.9945,Y -6.621,Z 80,A -10.7348,B 24.906,C -2.239,E1 25.1591,E2 95.3788} C_DIS
LIN {X 78.3837,Y -11.8322,Z 80,A -14.4366,B 24.9067,C -2.2298,E1 25.1578,E2 99.0806} C_DIS
LIN {X 77.7562,Y -15.426,Z 80,A -17.0719,B 24.9074,C -2.2215,E1 25.1564,E2 101.7202} C_DIS
LIN {X 77.1438,Y -18.2413,Z 80,A -19.1668,B 24.908,C -2.2145,E1 25.1551,E2 103.8193} C_DIS
LIN {X 76.274,Y -21.5916,Z 80,A -21.5123,B 24.9082,C -2.2116,E1 25.1534,E2 106.1582} C_DIS
LIN {X 75.4355,Y -24.3598,Z 80,A -23.7466,B 24.9092,C -2.2006,E1 25.1515,E2 108.4058} C_DIS
LIN {X 74.6151,Y -26.7661,Z 80,A -25.4643,B 24.9093,C -2.1987,E1 25.15,E2 110.1182} C_DIS
LIN {X 73.1821,Y -30.4666,Z 80,A -28.3966,B 24.9102,C -2.188,E1 25.1469,E2 113.0597} C_DIS
LIN {X 71.7331,Y -33.7399,Z 80,A -30.9951,B 24.9109,C -2.1799,E1 25.1439,E2 115.6632} C_DIS
LIN {X 70.2451,Y -36.7355,Z 80,A -33.2982,B 24.9112,C -2.1764,E1 25.141,E2 117.9624} C_DIS
LIN {X 68.2329,Y -40.3509,Z 80,A -36.1227,B 24.9114,C -2.1729,E1 25.1371,E2 120.7803} C_DIS
LIN {X 67.0906,Y -42.2238,Z 80,A -37.9349,B 24.9124,C -2.1614,E1 25.1344,E2 122.6107} C_DIS
LIN {X 65.209,Y -45.075,Z 80,A -40.3569,B 24.9128,C -2.156,E1 25.1306,E2 125.0334} C_DIS
LIN {X 63.2522,Y -47.7821,Z 80,A -42.796,B 24.9134,C -2.1487,E1 25.1266,E2 127.4779} C_DIS
LIN {X 61.1255,Y -50.4743,Z 80,A -45.199,B 24.9137,C -2.1446,E1 25.1224,E2 129.8795} C_DIS
LIN {X 58.9978,Y -52.9451,Z 80,A -47.567,B 24.9142,C -2.1383,E1 25.118,E2 132.2518} C_DIS
LIN {X 56.7351,Y -55.3642,Z 80,A -50.0546,B 24.9149,C -2.1295,E1 25.1132,E2 134.7494} C_DIS
LIN {X 54.3277,Y -57.7271,Z 80,A -52.3494,B 24.9151,C -2.1282,E1 25.1086,E2 137.0379} C_DIS
LIN {X 51.8911,Y -59.9276,Z 80,A -54.8608,B 24.9158,C -2.1185,E1 25.1033,E2 139.5622} C_DIS
LIN {X 48.9986,Y -62.3145,Z 80,A -57.2327,B 24.9155,C -2.1229,E1 25.0982,E2 141.9146} C_DIS
LIN {X 46.8017,Y -63.9807,Z 80,A -59.4426,B 24.9163,C -2.1122,E1 25.0932,E2 144.142} C_DIS
LIN {X 43.9571,Y -65.968,Z 80,A -61.9267,B 24.9167,C -2.1079,E1 25.0875,E2 146.6278} C_DIS
LIN {X 41.068,Y -67.8038,Z 80,A -64.3837,B 24.917,C -2.1038,E1 25.0816,E2 149.0867} C_DIS
LIN {X 38.1573,Y -69.4846,Z 80,A -66.8416,B 24.9174,C -2.0986,E1 25.0756,E2 151.5495} C_DIS
LIN {X 35.2349,Y -71.01,Z 80,A -69.0069,B 24.9172,C -2.1012,E1 25.0703,E2 153.7028} C_DIS
LIN {X 32.5171,Y -72.295,Z 80,A -71.2897,B 24.9177,C -2.0946,E1 25.0645,E2 155.9955} C_DIS
LIN {X 29.5232,Y -73.5694,Z 80,A -73.6716,B 24.9181,C -2.0903,E1 25.0583,E2 158.382} C_DIS
LIN {X 25.6741,Y -74.9993,Z 80,A -76.4857,B 24.9181,C -2.091,E1 25.0509,E2 161.1886} C_DIS
LIN {X 23.0145,Y -75.8563,Z 80,A -78.4129,B 24.918,C -2.0914,E1 25.0458,E2 163.1114} C_DIS
LIN {X 20.4152,Y -76.5977,Z 80,A -80.6248,B 24.9187,C -2.0817,E1 25.0398,E2 165.3427} C_DIS
LIN {X 17.3243,Y -77.3556,Z 80,A -82.9116,B 24.9189,C -2.0799,E1 25.0336,E2 167.6305} C_DIS
LIN {X 14.4819,Y -77.938,Z 80,A -85.1096,B 24.9192,C -2.0752,E1 25.0276,E2 169.837} C_DIS
LIN {X 10.9211,Y -78.5156,Z 80,A -87.5792,B 24.9191,C -2.0774,E1 25.0208,E2 172.2992} C_DIS
LIN {X 6.1536,Y -79.0318,Z 80,A -90.8713,B 24.9188,C -2.0805,E1 25.0116,E2 175.5818} C_DIS
LIN {X 3.3673,Y -79.1996,Z 80,A -93.065,B 24.9193,C -2.0746,E1 25.0055,E2 177.7886} C_DIS
LIN {X 0.5113,Y -79.2679,Z 80,A -94.2674,B 24.9174,C -2.0989,E1 25.0023,E2 178.9333} C_DIS
Enddeposition()
LIN {X 0.5113,Y -79.2679,Z 80,A -94.2674,B 24.9174,C -2.0989,E1 25.0023,E2 178.9333} C_DIS
Startdeposition()
$VEL.CP = VEL_PRINT
LIN {X 2.4537,Y -78.3387,Z 80,A -92.6304,B 24.9156,C -2.121,E1 25.007,E2 177.2442} C_DIS
LIN {X 6.2696,Y -78.1259,Z 80,A -89.7316,B 24.9153,C -2.1253,E1 25.0151,E2 174.3365} C_DIS
LIN {X 10.8231,Y -77.6265,Z 80,A -86.5597,B 24.9155,C -2.1221,E1 25.0239,E2 171.1744} C_DIS
LIN {X 15.2049,Y -76.8888,Z 80,A -83.28,B 24.9153,C -2.1256,E1 25.0329,E2 167.8901} C_DIS
LIN {X 18.3337,Y -76.2022,Z 80,A -80.9423,B 24.9151,C -2.1277,E1 25.0393,E2 165.5506} C_DIS
LIN {X 21.5607,Y -75.3535,Z 80,A -78.7332,B 24.9154,C -2.1235,E1 25.0452,E2 163.3551} C_DIS
LIN {X 25.1133,Y -74.2449,Z 80,A -76.0649,B 24.9153,C -2.1251,E1 25.0523,E2 160.6878} C_DIS
LIN {X 28.5014,Y -73.0115,Z 80,A -72.9326,B 24.9138,C -2.1435,E1 25.0606,E2 157.5187} C_DIS
LIN {X 32.1572,Y -71.4765,Z 80,A -70.2892,B 24.9141,C -2.1401,E1 25.0673,E2 154.8898} C_DIS
LIN {X 36.5755,Y -69.3195,Z 80,A -66.7191,B 24.9137,C -2.1452,E1 25.0762,E2 151.3172} C_DIS
LIN {X 39.3902,Y -67.7608,Z 80,A -64.2747,B 24.9131,C -2.1521,E1 25.0822,E2 148.8637} C_DIS
LIN {X 42.324,Y -65.967,Z 80,A -61.8021,B 24.9128,C -2.1556,E1 25.088,E2 146.3906} C_DIS
LIN {X 45.1217,Y -64.0865,Z 80,A -59.1732,B 24.912,C -2.1656,E1 25.0941,E2 143.7472} C_DIS
LIN {X 48.331,Y -61.7026,Z 80,A -56.7736,B 24.9128,C -2.1557,E1 25.0994,E2 141.3797} C_DIS
LIN {X 49.948,Y -60.4004,Z 80,A -54.9233,B 24.9117,C -2.1693,E1 25.1034,E2 139.5044} C_DIS
LIN {X 52.4243,Y -58.2641,Z 80,A -52.5986,B 24.9115,C -2.1727,E1 25.1083,E2 137.1808} C_DIS
LIN {X 54.2222,Y -56.5949,Z 80,A -50.8736,B 24.9113,C -2.1748,E1 25.1118,E2 135.458} C_DIS
LIN {X 56.4046,Y -54.4196,Z 80,A -48.5905,B 24.9108,C -2.1812,E1 25.1163,E2 133.1694} C_DIS
LIN {X 58.708,Y -51.9272,Z 80,A -46.0628,B 24.9101,C -2.1889,E1 25.121,E2 130.6348} C_DIS
LIN {X 61.1775,Y -48.9946,Z 80,A -43.3257,B 24.9097,C -2.1941,E1 25.1259,E2 127.8979} C_DIS
LIN {X 63.3462,Y -46.1549,Z 80,A -40.6822,B 24.909,C -2.2021,E1 25.1303,E2 125.2481} C_DIS
LIN {X 65.2019,Y -43.4946,Z 80,A -38.3162,B 24.9085,C -2.2085,E1 25.134,E2 122.8788} C_DIS
LIN {X 66.736,Y -41.1029,Z 80,A -36.0985,B 24.9077,C -2.2188,E1 25.1373,E2 120.6481} C_DIS
LIN {X 69.0407,Y -37.1001,Z 80,A -32.5348,B 24.9063,C -2.2344,E1 25.1422,E2 117.0659} C_DIS
LIN {X 71.0236,Y -33.1455,Z 80,A -29.8846,B 24.9071,C -2.2256,E1 25.1454,E2 114.4508} C_DIS
LIN {X 73.2862,Y -27.7867,Z 80,A -25.489,B 24.9056,C -2.2429,E1 25.1501,E2 110.0385} C_DIS
LIN {X 74.6772,Y -23.7994,Z 80,A -22.3775,B 24.9048,C -2.2532,E1 25.1528,E2 106.9202} C_DIS
LIN {X 75.6292,Y -20.5724,Z 80,A -20.0313,B 24.9044,C -2.2573,E1 25.1546,E2 104.5778} C_DIS
LIN {X 76.4089,Y -17.4554,Z 80,A -17.8246,B 24.9042,C -2.2602,E1 25.156,E2 102.377} C_DIS
LIN {X 77.2573,Y -13.2044,Z 80,A -14.8515,B 24.9038,C -2.2641,E1 25.1576,E2 99.4123} C_DIS
LIN {X 77.6165,Y -10.8939,Z 80,A -12.4271,B 24.9014,C -2.2922,E1 25.1586,E2 96.9358} C_DIS
LIN {X 78.256,Y -4.3559,Z 80,A -8.4149,B 24.9023,C -2.2824,E1 25.1596,E2 92.9703} C_DIS
LIN {X 78.3757,Y 0.431,Z 80,A -5.0963,B 24.9018,C -2.2878,E1 25.1598,E2 89.6587} C_DIS
LIN {X 78.2486,Y 4.4892,Z 80,A -1.6753,B 24.8998,C -2.3114,E1 25.1594,E2 86.2023} C_DIS
LIN {X 78.0533,Y 7.1164,Z 80,A 0.4885,B 24.8986,C -2.325,E1 25.1589,E2 84.0192} C_DIS
LIN {X 77.5666,Y 11.2448,Z 80,A 3.6425,B 24.8974,C -2.3382,E1 25.1577,E2 80.8528} C_DIS
LIN {X 76.9099,Y 15.0974,Z 80,A 5.9707,B 24.8981,C -2.3303,E1 25.1566,E2 78.5568} C_DIS
LIN {X 76.2995,Y 17.9282,Z 80,A 8.2752,B 24.897,C -2.3427,E1 25.1552,E2 76.2364} C_DIS
LIN {X 75.54,Y 20.8952,Z 80,A 10.4152,B 24.8967,C -2.3464,E1 25.1536,E2 74.1001} C_DIS
LIN {X 74.7873,Y 23.4499,Z 80,A 12.5695,B 24.8956,C -2.3587,E1 25.1518,E2 71.929} C_DIS
LIN {X 73.8796,Y 26.1684,Z 80,A 15.649,B 24.8923,C -2.3959,E1 25.1489,E2 68.7788} C_DIS
LIN {X 72.071,Y 30.801,Z 80,A 17.8187,B 24.8955,C -2.3602,E1 25.1467,E2 66.7054} C_DIS
LIN {X 69.8735,Y 35.5064,Z 80,A 21.9295,B 24.8937,C -2.3805,E1 25.1417,E2 62.5688} C_DIS
LIN {X 68.3991,Y 38.2694,Z 80,A 24.685,B 24.8918,C -2.4011,E1 25.1379,E2 59.7788} C_DIS
LIN {X 65.8983,Y 42.4312,Z 80,A 27.7376,B 24.8924,C -2.3949,E1 25.1335,E2 56.7564} C_DIS
LIN {X 64.3962,Y 44.6779,Z 80,A 29.8448,B 24.8916,C -2.4039,E1 25.1301,E2 54.6383} C_DIS
LIN {X 61.436,Y 48.6683,Z 80,A 33.2651,B 24.8914,C -2.4061,E1 25.1243,E2 51.229} C_DIS
LIN {X 59.867,Y 50.5868,Z 80,A 35.1555,B 24.8908,C -2.4127,E1 25.1209,E2 49.3318} C_DIS
LIN {X 57.2786,Y 53.4997,Z 80,A 38.1027,B 24.8899,C -2.422,E1 25.1154,E2 46.3755} C_DIS
LIN {X 54.4593,Y 56.3664,Z 80,A 40.6145,B 24.8905,C -2.4152,E1 25.1105,E2 43.8904} C_DIS
LIN {X 52.5867,Y 58.1178,Z 80,A 42.7192,B 24.8896,C -2.4259,E1 25.1061,E2 41.7689} C_DIS
LIN {X 50.1027,Y 60.2719,Z 80,A 44.9485,B 24.8896,C -2.4253,E1 25.1014,E2 39.5498} C_DIS
LIN {X 47.0739,Y 62.6659,Z 80,A 48.3471,B 24.8876,C -2.4476,E1 25.0938,E2 36.1108} C_DIS
LIN {X 43.2886,Y 65.3383,Z 80,A 51.315,B 24.8882,C -2.4406,E1 25.087,E2 33.1696} C_DIS
LIN {X 40.6372,Y 67.0194,Z 80,A 53.6737,B 24.8877,C -2.4459,E1 25.0814,E2 30.8057} C_DIS
LIN {X 37.4549,Y 68.8485,Z 80,A 56.088,B 24.8881,C -2.4417,E1 25.0755,E2 28.4086} C_DIS
LIN {X 33.4755,Y 70.8692,Z 80,A 59.5689,B 24.8872,C -2.4521,E1 25.0668,E2 24.9124} C_DIS
LIN {X 29.5645,Y 72.5873,Z 80,A 62.4412,B 24.8875,C -2.4481,E1 25.0595,E2 22.0563} C_DIS
LIN {X 26.0244,Y 73.9305,Z 80,A 65.3323,B 24.887,C -2.4542,E1 25.0519,E2 19.1568} C_DIS
LIN {X 23.9975,Y 74.6131,Z 80,A 67.1001,B 24.8863,C -2.4614,E1 25.0471,E2 17.3754} C_DIS
LIN {X 20.1493,Y 75.7435,Z 80,A 69.8797,B 24.8865,C -2.4589,E1 25.0397,E2 14.6062} C_DIS
LIN {X 16.9243,Y 76.5284,Z 80,A 71.9522,B 24.8873,C -2.4501,E1 25.0341,E2 12.5575} C_DIS
LIN {X 14.9367,Y 76.9408,Z 80,A 73.8238,B 24.8863,C -2.4618,E1 25.0289,E2 10.6604} C_DIS
LIN {X 12.4707,Y 77.3799,Z 80,A 75.7027,B 24.8861,C -2.4637,E1 25.0237,E2 8.7788} C_DIS
LIN {X 9.2388,Y 77.8305,Z 80,A 78.2635,B 24.8856,C -2.4692,E1 25.0166,E2 6.207} C_DIS
LIN {X 4.0083,Y 78.2746,Z 80,A 81.6087,B 24.8868,C -2.4555,E1 25.0074,E2 2.896} C_DIS
LIN {X 0.8011,Y 78.3728,Z 80,A 84.1944,B 24.8862,C -2.4619,E1 25.0001,E2 0.2956} C_DIS
LIN {X -2.4185,Y 78.3396,Z 80,A 86.5409,B 24.8863,C -2.4611,E1 24.9936,E2 -2.0492} C_DIS
LIN {X -6.0743,Y 78.1412,Z 80,A 89.2521,B 24.8863,C -2.461,E1 24.986,E2 -4.7611} C_DIS
LIN {X -9.4958,Y 77.7996,Z 80,A 91.6581,B 24.8867,C -2.4566,E1 24.9794,E2 -7.1582} C_DIS
LIN {X -12.2901,Y 77.4082,Z 80,A 93.8038,B 24.8867,C -2.4575,E1 24.9734,E2 -9.3079} C_DIS
LIN {X -15.0077,Y 76.9271,Z 80,A 95.7865,B 24.8869,C -2.455,E1 24.968,E2 -11.2868} C_DIS
LIN {X -19.4966,Y 75.9135,Z 80,A 99.1711,B 24.8871,C -2.4525,E1 24.9588,E2 -14.6698} C_DIS
LIN {X -22.3364,Y 75.127,Z 80,A 101.3924,B 24.8871,C -2.452,E1 24.9528,E2 -16.8935} C_DIS
LIN {X -29.062,Y 72.7909,Z 80,A 106.4325,B 24.8882,C -2.4409,E1 24.9397,E2 -21.9175} C_DIS
LIN {X -32.2877,Y 71.4177,Z 80,A 109.3799,B 24.8876,C -2.4474,E1 24.9321,E2 -24.8874} C_DIS
LIN {X -35.854,Y 69.6958,Z 80,A 112.8639,B 24.8866,C -2.4584,E1 24.9233,E2 -28.4069} C_DIS
LIN {X -39.3954,Y 67.7578,Z 80,A 115.0562,B 24.8889,C -2.4332,E1 24.9181,E2 -30.5455} C_DIS
LIN {X -42.2403,Y 66.0208,Z 80,A 117.4591,B 24.8894,C -2.4278,E1 24.9124,E2 -32.9432} C_DIS
LIN {X -44.8307,Y 64.29,Z 80,A 120.2001,B 24.8887,C -2.4354,E1 24.9061,E2 -35.7116} C_DIS
LIN {X -48.9935,Y 61.1783,Z 80,A 123.6225,B 24.8903,C -2.4176,E1 24.8986,E2 -39.1041} C_DIS
LIN {X -51.6589,Y 58.9437,Z 80,A 126.1436,B 24.8909,C -2.4114,E1 24.8932,E2 -41.6202} C_DIS
LIN {X -53.7275,Y 57.0643,Z 80,A 128.3709,B 24.8909,C -2.4114,E1 24.8887,E2 -43.8567} C_DIS
LIN {X -57.2009,Y 53.5822,Z 80,A 131.7803,B 24.8921,C -2.398,E1 24.8821,E2 -47.2486} C_DIS
LIN {X -59.3803,Y 51.1569,Z 80,A 134.1416,B 24.8927,C -2.3914,E1 24.8777,E2 -49.6049} C_DIS
LIN {X -60.8337,Y 49.4191,Z 80,A 136.2047,B 24.8921,C -2.3975,E1 24.8741,E2 -51.692} C_DIS
LIN {X -63.7991,Y 45.5264,Z 80,A 139.865,B 24.8928,C -2.39,E1 24.868,E2 -55.3522} C_DIS
LIN {X -66.3189,Y 41.7715,Z 80,A 142.7895,B 24.8945,C -2.3712,E1 24.8636,E2 -58.2464} C_DIS
LIN {X -69.7793,Y 35.6907,Z 80,A 147.8028,B 24.896,C -2.3539,E1 24.8568,E2 -63.2448} C_DIS
LIN {X -71.322,Y 32.4989,Z 80,A 150.1236,B 24.8973,C -2.3395,E1 24.8541,E2 -65.5438} C_DIS
LIN {X -73.1436,Y 28.1624,Z 80,A 153.8668,B 24.8976,C -2.3366,E1 24.8501,E2 -69.301} C_DIS
LIN {X -74.4071,Y 24.6266,Z 80,A 157.2069,B 24.897,C -2.3431,E1 24.847,E2 -72.6756} C_DIS
LIN {X -76.2458,Y 18.152,Z 80,A 161.7631,B 24.8991,C -2.3186,E1 24.8437,E2 -77.1997} C_DIS
LIN {X -76.9641,Y 14.8158,Z 80,A 164.2326,B 24.8999,C -2.3101,E1 24.8424,E2 -79.6635} C_DIS
LIN {X -77.475,Y 11.8582,Z 80,A 166.475,B 24.9004,C -2.3043,E1 24.8414,E2 -81.9055} C_DIS
LIN {X -77.8759,Y 8.8534,Z 80,A 168.716,B 24.9009,C -2.2979,E1 24.8406,E2 -84.1445} C_DIS
LIN {X -78.1875,Y 5.4513,Z 80,A 171.2379,B 24.9016,C -2.2906,E1 24.8401,E2 -86.664} C_DIS
LIN {X -78.3486,Y 2.1014,Z 80,A 173.6503,B 24.9023,C -2.2818,E1 24.8398,E2 -89.07} C_DIS
LIN {X -78.3677,Y -1.2328,Z 80,A 175.8923,B 24.9034,C -2.2692,E1 24.8398,E2 -91.2954} C_DIS
LIN {X -78.2731,Y -4.0367,Z 80,A 178.4179,B 24.9029,C -2.2745,E1 24.8401,E2 -93.849} C_DIS
LIN {X -77.9658,Y -8.0206,Z 80,A -178.8924,B 24.9042,C -2.2595,E1 24.8408,E2 -96.519} C_DIS
LIN {X -77.5763,Y -11.1769,Z 80,A -176.9056,B 24.9055,C -2.2439,E1 24.8415,E2 -98.4803} C_DIS
LIN {X -77.2068,Y -13.4978,Z 80,A -174.5341,B 24.9046,C -2.2549,E1 24.8426,E2 -100.8922} C_DIS
LIN {X -76.402,Y -17.4851,Z 80,A -171.8059,B 24.9059,C -2.2396,E1 24.8442,E2 -103.5999} C_DIS
LIN {X -75.6456,Y -20.5114,Z 80,A -168.6509,B 24.9046,C -2.2549,E1 24.8466,E2 -106.8098} C_DIS
LIN {X -74.456,Y -24.479,Z 80,A -165.8765,B 24.9059,C -2.2394,E1 24.849,E2 -109.5632} C_DIS
LIN {X -73.3306,Y -27.6697,Z 80,A -164.1342,B 24.9081,C -2.2137,E1 24.8506,E2 -111.2539} C_DIS
LIN {X -72.1796,Y -30.5466,Z 80,A -161.6803,B 24.9082,C -2.212,E1 24.8532,E2 -113.7173} C_DIS
LIN {X -70.754,Y -33.7182,Z 80,A -159.1932,B 24.9089,C -2.2035,E1 24.8561,E2 -116.1978} C_DIS
LIN {X -69.8332,Y -35.5851,Z 80,A -157.6331,B 24.9092,C -2.2003,E1 24.8581,E2 -117.7586} C_DIS
LIN {X -66.79,Y -41.0147,Z 80,A -153.0006,B 24.91,C -2.1903,E1 24.8645,E2 -122.3914} C_DIS
LIN {X -63.6278,Y -45.7664,Z 80,A -148.8226,B 24.9109,C -2.18,E1 24.8711,E2 -126.5655} C_DIS
LIN {X -61.6243,Y -48.43,Z 80,A -146.4037,B 24.9114,C -2.1737,E1 24.8752,E2 -128.9809} C_DIS
LIN {X -59.6989,Y -50.7841,Z 80,A -144.3693,B 24.9122,C -2.1637,E1 24.8788,E2 -131.0008} C_DIS
LIN {X -57.1884,Y -53.5955,Z 80,A -141.5108,B 24.9125,C -2.1603,E1 24.8842,E2 -133.8639} C_DIS
LIN {X -54.6896,Y -56.1444,Z 80,A -138.688,B 24.9125,C -2.1604,E1 24.8898,E2 -136.6989} C_DIS
LIN {X -52.0555,Y -58.594,Z 80,A -136.0892,B 24.9129,C -2.1544,E1 24.8952,E2 -139.2939} C_DIS
LIN {X -49.725,Y -60.5847,Z 80,A -133.1576,B 24.9118,C -2.1687,E1 24.9016,E2 -142.2706} C_DIS
LIN {X -46.7967,Y -62.8742,Z 80,A -131.1245,B 24.9137,C -2.1456,E1 24.906,E2 -144.2561} C_DIS
LIN {X -44.107,Y -64.7888,Z 80,A -128.4663,B 24.9134,C -2.1483,E1 24.9121,E2 -146.9296} C_DIS
LIN {X -40.75,Y -66.9508,Z 80,A -125.7886,B 24.9143,C -2.1374,E1 24.9184,E2 -149.5899} C_DIS
LIN {X -36.2377,Y -69.4966,Z 80,A -121.2967,B 24.9132,C -2.1516,E1 24.9296,E2 -154.1283} C_DIS
LIN {X -32.96,Y -71.1095,Z 80,A -119.5325,B 24.9154,C -2.1237,E1 24.9339,E2 -155.8306} C_DIS
LIN {X -31.0765,Y -71.9521,Z 80,A -117.6622,B 24.9147,C -2.132,E1 24.9387,E2 -157.725} C_DIS
LIN {X -27.7192,Y -73.3118,Z 80,A -115.4772,B 24.916,C -2.1168,E1 24.9443,E2 -159.8785} C_DIS
LIN {X -25.2604,Y -74.1953,Z 80,A -113.2657,B 24.9154,C -2.1235,E1 24.9502,E2 -162.1102} C_DIS
LIN {X -21.8807,Y -75.2622,Z 80,A -110.5624,B 24.9154,C -2.1247,E1 24.9574,E2 -164.8212} C_DIS
LIN {X -19.1308,Y -76.006,Z 80,A -108.7022,B 24.9159,C -2.1174,E1 24.9624,E2 -166.6667} C_DIS
LIN {X -16.0603,Y -76.7146,Z 80,A -106.0623,B 24.9153,C -2.1257,E1 24.9697,E2 -169.3297} C_DIS
LIN {X -12.3674,Y -77.3962,Z 80,A -103.3466,B 24.9153,C -2.124,E1 24.9772,E2 -172.044} C_DIS
LIN {X -8.0436,Y -77.9634,Z 80,A -100.353,B 24.9159,C -2.1181,E1 24.9854,E2 -175.0254} C_DIS
LIN {X -1.9985,Y -78.3514,Z 80,A -95.9998,B 24.916,C -2.1161,E1 24.9976,E2 -179.3752} C_DIS
LIN {X 0.5009,Y -78.3613,Z 80,A -94.3406,B 24.9164,C -2.1119,E1 25.0022,E2 -181.0245} C_DIS
Enddeposition()
LIN {X 0.5009,Y -78.3613,Z 80,A -94.3406,B 24.9164,C -2.1119,E1 25.0022,E2 -181.0245} C_DIS
Startdeposition()
$VEL.CP = VEL_PRINT
LIN {X -0.5198,Y -77.4813,Z 80,A -95.9279,B 24.917,C -2.1036,E1 24.9977,E2 -179.4175} C_DIS
LIN {X -5.8722,Y -77.2599,Z 80,A -99.7744,B 24.9168,C -2.1065,E1 24.987,E2 -175.5769} C_DIS
LIN {X -9.8256,Y -76.8577,Z 80,A -103.1105,B 24.9176,C -2.096,E1 24.9776,E2 -172.2137} C_DIS
LIN {X -13.5293,Y -76.2923,Z 80,A -105.6944,B 24.9171,C -2.1019,E1 24.9705,E2 -169.6415} C_DIS
LIN {X -15.8048,Y -75.8544,Z 80,A -107.4152,B 24.9171,C -2.1024,E1 24.9658,E2 -167.9198} C_DIS
LIN {X -19.6939,Y -74.9393,Z 80,A -110.3975,B 24.9171,C -2.1032,E1 24.9577,E2 -164.9353} C_DIS
LIN {X -23.1348,Y -73.9489,Z 80,A -112.8909,B 24.9166,C -2.1092,E1 24.9511,E2 -162.4519} C_DIS
LIN {X -26.9122,Y -72.6587,Z 80,A -115.5809,B 24.9158,C -2.1187,E1 24.9441,E2 -159.7792} C_DIS
LIN {X -29.2555,Y -71.7473,Z 80,A -117.897,B 24.9166,C -2.1083,E1 24.938,E2 -157.4334} C_DIS
LIN {X -32.3302,Y -70.4153,Z 80,A -120.0432,B 24.9157,C -2.1198,E1 24.9326,E2 -155.3093} C_DIS
LIN {X -36.0185,Y -68.6021,Z 80,A -123.6841,B 24.9167,C -2.1078,E1 24.9234,E2 -151.6301} C_DIS
LIN {X -39.8348,Y -66.4602,Z 80,A -126.6836,B 24.9158,C -2.1184,E1 24.9162,E2 -148.6469} C_DIS
LIN {X -44.3391,Y -63.5428,Z 80,A -130.3245,B 24.9147,C -2.1331,E1 24.9078,E2 -145.0291} C_DIS
LIN {X -47.3949,Y -61.2974,Z 80,A -133.7486,B 24.9155,C -2.1221,E1 24.9,E2 -141.5664} C_DIS
LIN {X -50.8056,Y -58.5018,Z 80,A -136.6779,B 24.9144,C -2.1366,E1 24.8938,E2 -138.6605} C_DIS
LIN {X -53.3668,Y -56.176,Z 80,A -139.6544,B 24.9148,C -2.1312,E1 24.8877,E2 -135.6589} C_DIS
LIN {X -56.6133,Y -52.902,Z 80,A -143.4182,B 24.9149,C -2.1297,E1 24.8804,E2 -131.8752} C_DIS
LIN {X -59.1951,Y -49.9967,Z 80,A -145.5535,B 24.9129,C -2.1546,E1 24.8766,E2 -129.7895} C_DIS
LIN {X -61.3112,Y -47.377,Z 80,A -148.0179,B 24.9124,C -2.1611,E1 24.8724,E2 -127.3291} C_DIS
LIN {X -64.6527,Y -42.7037,Z 80,A -152.0586,B 24.9111,C -2.1768,E1 24.8659,E2 -123.3059} C_DIS
LIN {X -65.8372,Y -40.8547,Z 80,A -154.1585,B 24.9117,C -2.1692,E1 24.8628,E2 -121.1772} C_DIS
LIN {X -68.0388,Y -37.0726,Z 80,A -157.461,B 24.9112,C -2.1762,E1 24.8582,E2 -117.8742} C_DIS
LIN {X -69.6988,Y -33.8496,Z 80,A -159.8981,B 24.9101,C -2.1895,E1 24.8552,E2 -115.4557} C_DIS
LIN {X -71.044,Y -30.9253,Z 80,A -162.6971,B 24.9104,C -2.1861,E1 24.852,E2 -112.633} C_DIS
LIN {X -72.6011,Y -27.0668,Z 80,A -165.562,B 24.9092,C -2.2001,E1 24.8492,E2 -109.7855} C_DIS
LIN {X -73.5958,Y -24.2326,Z 80,A -167.7613,B 24.9086,C -2.2071,E1 24.8472,E2 -107.5905} C_DIS
LIN {X -74.9289,Y -19.7337,Z 80,A -171.0224,B 24.9073,C -2.2226,E1 24.8447,E2 -104.3474} C_DIS
LIN {X -75.6327,Y -16.8347,Z 80,A -173.933,B 24.9082,C -2.2124,E1 24.8429,E2 -101.3953} C_DIS
LIN {X -76.2869,Y -13.5634,Z 80,A -176.1631,B 24.9071,C -2.2257,E1 24.8418,E2 -99.1837} C_DIS
LIN {X -76.8028,Y -10.249,Z 80,A -178.2915,B 24.9057,C -2.2418,E1 24.841,E2 -97.0812} C_DIS
LIN {X -77.1576,Y -7.095,Z 80,A 178.7548,B 24.9063,C -2.2347,E1 24.8402,E2 -94.0928} C_DIS
LIN {X -77.3896,Y -3.8169,Z 80,A 176.5431,B 24.9052,C -2.2476,E1 24.8399,E2 -91.8985} C_DIS
LIN {X -77.4837,Y 0.0597,Z 80,A 173.9752,B 24.9039,C -2.2638,E1 24.8398,E2 -89.3539} C_DIS
LIN {X -77.4101,Y 3.3612,Z 80,A 171.5056,B 24.9032,C -2.2709,E1 24.84,E2 -86.8865} C_DIS
LIN {X -77.142,Y 7.2611,Z 80,A 168.2742,B 24.9032,C -2.272,E1 24.8408,E2 -83.6383} C_DIS
LIN {X -76.7268,Y 10.8,Z 80,A 165.9699,B 24.9018,C -2.2883,E1 24.8416,E2 -81.359} C_DIS
LIN {X -76.236,Y 13.846,Z 80,A 163.7316,B 24.9011,C -2.2965,E1 24.8426,E2 -79.1271} C_DIS
LIN {X -75.4577,Y 17.6007,Z 80,A 160.7644,B 24.9006,C -2.3023,E1 24.8444,E2 -76.1563} C_DIS
LIN {X -74.5002,Y 21.2927,Z 80,A 157.8393,B 24.9,C -2.3086,E1 24.8465,E2 -73.2292} C_DIS
LIN {X -72.813,Y 26.4934,Z 80,A 154.1172,B 24.8982,C -2.3287,E1 24.8498,E2 -69.534} C_DIS
LIN {X -72.105,Y 28.3637,Z 80,A 151.7699,B 24.8997,C -2.3124,E1 24.8523,E2 -67.1346} C_DIS
LIN {X -70.7588,Y 31.5738,Z 80,A 150.1887,B 24.8969,C -2.3439,E1 24.854,E2 -65.6199} C_DIS
LIN {X -69.2058,Y 34.8463,Z 80,A 147.4326,B 24.8964,C -2.3499,E1 24.8573,E2 -62.8632} C_DIS
LIN {X -67.5396,Y 37.9747,Z 80,A 144.1054,B 24.8972,C -2.3404,E1 24.8618,E2 -59.4958} C_DIS
LIN {X -65.3397,Y 41.6463,Z 80,A 141.2578,B 24.8958,C -2.357,E1 24.8659,E2 -56.6731} C_DIS
LIN {X -62.805,Y 45.3802,Z 80,A 138.183,B 24.8944,C -2.3725,E1 24.8708,E2 -53.62} C_DIS
LIN {X -59.7727,Y 49.3045,Z 80,A 134.2592,B 24.8941,C -2.3758,E1 24.8776,E2 -49.6857} C_DIS
LIN {X -57.6676,Y 51.7502,Z 80,A 131.0906,B 24.8952,C -2.3627,E1 24.8836,E2 -46.4717} C_DIS
LIN {X -55.0575,Y 54.5189,Z 80,A 129.0438,B 24.893,C -2.3882,E1 24.8874,E2 -44.477} C_DIS
LIN {X -52.6075,Y 56.8873,Z 80,A 126.4335,B 24.8926,C -2.3919,E1 24.8927,E2 -41.8646} C_DIS
LIN {X -49.9079,Y 59.2706,Z 80,A 123.6995,B 24.8923,C -2.396,E1 24.8985,E2 -39.1299} C_DIS
LIN {X -47.0796,Y 61.5401,Z 80,A 120.1186,B 24.8938,C -2.3795,E1 24.9066,E2 -35.4964} C_DIS
LIN {X -43.4445,Y 64.1577,Z 80,A 117.968,B 24.8906,C -2.4149,E1 24.9113,E2 -33.4229} C_DIS
LIN {X -40.275,Y 66.1933,Z 80,A 114.8968,B 24.8907,C -2.4128,E1 24.9186,E2 -30.3371} C_DIS
LIN {X -37.4132,Y 67.8529,Z 80,A 112.5416,B 24.8902,C -2.4193,E1 24.9243,E2 -27.9906} C_DIS
LIN {X -34.905,Y 69.1762,Z 80,A 110.5552,B 24.8896,C -2.4256,E1 24.9292,E2 -26.0136} C_DIS
LIN {X -31.78,Y 70.6659,Z 80,A 107.5387,B 24.8903,C -2.4178,E1 24.9369,E2 -22.9712} C_DIS
LIN {X -28.784,Y 71.9395,Z 80,A 104.9894,B 24.8903,C -2.4175,E1 24.9436,E2 -20.4154} C_DIS
LIN {X -23.5274,Y 73.8255,Z 80,A 101.2398,B 24.889,C -2.4323,E1 24.9534,E2 -16.6938} C_DIS
LIN {X -19.0457,Y 75.1054,Z 80,A 97.7076,B 24.8889,C -2.4336,E1 24.9629,E2 -13.1594} C_DIS
LIN {X -14.7523,Y 76.0658,Z 80,A 94.7745,B 24.8878,C -2.4448,E1 24.9708,E2 -10.2493} C_DIS
LIN {X -11.9779,Y 76.5518,Z 80,A 92.5658,B 24.888,C -2.4429,E1 24.9769,E2 -8.0341} C_DIS
LIN {X -8.8353,Y 76.9778,Z 80,A 89.9796,B 24.8885,C -2.4379,E1 24.9842,E2 -5.4342} C_DIS
LIN {X -5.5341,Y 77.2854,Z 80,A 87.3407,B 24.8888,C -2.434,E1 24.9915,E2 -2.7849} C_DIS
LIN {X -0.7193,Y 77.4801,Z 80,A 83.7005,B 24.8889,C -2.4329,E1 25.0017,E2 0.8582} C_DIS
LIN {X 2.8034,Y 77.432,Z 80,A 81.4394,B 24.888,C -2.4425,E1 25.008,E2 3.0963} C_DIS
LIN {X 6.9514,Y 77.1708,Z 80,A 78.2873,B 24.8882,C -2.4402,E1 25.0167,E2 6.2522} C_DIS
LIN {X 11.7247,Y 76.5909,Z 80,A 75.3686,B 24.8867,C -2.4569,E1 25.0247,E2 9.1289} C_DIS
LIN {X 14.5714,Y 76.1006,Z 80,A 72.633,B 24.8883,C -2.4395,E1 25.0323,E2 11.9027} C_DIS
LIN {X 18.0627,Y 75.3478,Z 80,A 70.1599,B 24.888,C -2.4428,E1 25.039,E2 14.3646} C_DIS
LIN {X 21.2882,Y 74.5015,Z 80,A 67.2905,B 24.8892,C -2.43,E1 25.0468,E2 17.2597} C_DIS
LIN {X 24.875,Y 73.3817,Z 80,A 64.8212,B 24.8886,C -2.4364,E1 25.0533,E2 19.7092} C_DIS
LIN {X 28.5572,Y 72.0289,Z 80,A 61.9563,B 24.8888,C -2.4346,E1 25.0608,E2 22.5721} C_DIS
LIN {X 33.2394,Y 69.9919,Z 80,A 57.7865,B 24.8902,C -2.4193,E1 25.0715,E2 26.7679} C_DIS
LIN {X 36.8582,Y 68.155,Z 80,A 55.1487,B 24.8896,C -2.4257,E1 25.0779,E2 29.3831} C_DIS
LIN {X 40.9912,Y 65.7522,Z 80,A 51.8714,B 24.8894,C -2.4279,E1 25.0858,E2 32.645} C_DIS
LIN {X 43.4341,Y 64.1647,Z 80,A 48.683,B 24.8924,C -2.3948,E1 25.0933,E2 35.9011} C_DIS
LIN {X 46.8551,Y 61.7116,Z 80,A 46.3027,B 24.891,C -2.4104,E1 25.0985,E2 38.2358} C_DIS
LIN {X 49.5224,Y 59.5916,Z 80,A 44.0082,B 24.8908,C -2.4123,E1 25.1035,E2 40.5172} C_DIS
LIN {X 51.9332,Y 57.5034,Z 80,A 41.5623,B 24.8914,C -2.4051,E1 25.1086,E2 42.9704} C_DIS
LIN {X 53.9931,Y 55.574,Z 80,A 39.1325,B 24.8927,C -2.3908,E1 25.1135,E2 45.424} C_DIS
LIN {X 57.4261,Y 52.0186,Z 80,A 35.5195,B 24.8933,C -2.384,E1 25.1204,E2 49.0372} C_DIS
LIN {X 59.6766,Y 49.4201,Z 80,A 33.4018,B 24.8927,C -2.3907,E1 25.1242,E2 51.1294} C_DIS
LIN {X 62.9851,Y 45.1279,Z 80,A 29.4828,B 24.8934,C -2.3837,E1 25.1308,E2 55.0463} C_DIS
LIN {X 64.3482,Y 43.1631,Z 80,A 27.5707,B 24.8942,C -2.3749,E1 25.1338,E2 56.9698} C_DIS
LIN {X 67.7159,Y 37.6591,Z 80,A 23.1071,B 24.8945,C -2.3717,E1 25.1402,E2 61.4182} C_DIS
LIN {X 68.977,Y 35.2959,Z 80,A 20.4954,B 24.8966,C -2.3473,E1 25.1436,E2 64.0737} C_DIS
LIN {X 70.7256,Y 31.6474,Z 80,A 18.1564,B 24.8956,C -2.3586,E1 25.1463,E2 66.3734} C_DIS
LIN {X 71.8604,Y 28.9788,Z 80,A 15.217,B 24.8983,C -2.3284,E1 25.1495,E2 69.3678} C_DIS
LIN {X 73.0295,Y 25.8905,Z 80,A 13.8039,B 24.8962,C -2.3525,E1 25.1508,E2 70.7161} C_DIS
LIN {X 74.0705,Y 22.7407,Z 80,A 10.9613,B 24.8978,C -2.3333,E1 25.1532,E2 73.588} C_DIS
LIN {X 74.9921,Y 19.4899,Z 80,A 8.4129,B 24.8986,C -2.3242,E1 25.1551,E2 76.1431} C_DIS
LIN {X 75.8309,Y 15.9187,Z 80,A 5.7628,B 24.8992,C -2.3178,E1 25.1567,E2 78.7929} C_DIS
LIN {X 76.3536,Y 13.1879,Z 80,A 3.513,B 24.9003,C -2.3056,E1 25.1578,E2 81.0585} C_DIS
LIN {X 76.9969,Y 8.6641,Z 80,A 0.0023,B 24.9015,C -2.291,E1 25.1591,E2 84.583} C_DIS
LIN {X 77.3004,Y 5.3183,Z 80,A -2.5108,B 24.9023,C -2.2822,E1 25.1596,E2 87.1018} C_DIS
LIN {X 77.4805,Y 0.6377,Z 80,A -5.5861,B 24.9023,C -2.2831,E1 25.1598,E2 90.1567} C_DIS
LIN {X 77.4166,Y -3.212,Z 80,A -7.9704,B 24.9018,C -2.2883,E1 25.1596,E2 92.5146} C_DIS
LIN {X 77.2889,Y -5.4865,Z 80,A -10.3784,B 24.9041,C -2.2607,E1 25.1592,E2 94.9735} C_DIS
LIN {X 76.842,Y -9.9467,Z 80,A -13.5732,B 24.9047,C -2.2538,E1 25.1581,E2 98.1657} C_DIS
LIN {X 76.3897,Y -12.972,Z 80,A -16.5178,B 24.9071,C -2.2258,E1 25.1568,E2 101.1591} C_DIS
LIN {X 75.5417,Y -17.2372,Z 80,A -18.5455,B 24.9049,C -2.2519,E1 25.1556,E2 103.1133} C_DIS
LIN {X 74.9427,Y -19.6806,Z 80,A -20.6757,B 24.9061,C -2.2378,E1 25.1541,E2 105.2646} C_DIS
LIN {X 74.0092,Y -22.9405,Z 80,A -23.8735,B 24.9085,C -2.2089,E1 25.1515,E2 108.5123} C_DIS
LIN {X 72.7825,Y -26.577,Z 80,A -25.645,B 24.9065,C -2.2328,E1 25.1499,E2 110.2176} C_DIS
LIN {X 70.8626,Y -31.3384,Z 80,A -29.6209,B 24.9079,C -2.2157,E1 25.1456,E2 114.2117} C_DIS
LIN {X 69.6463,Y -33.9547,Z 80,A -32.4142,B 24.9101,C -2.1893,E1 25.1422,E2 117.0524} C_DIS
LIN {X 68.103,Y -36.9541,Z 80,A -34.2041,B 24.9089,C -2.2035,E1 25.1399,E2 118.7996} C_DIS
LIN {X 65.7758,Y -40.9534,Z 80,A -37.523,B 24.9095,C -2.1968,E1 25.1352,E2 122.1171} C_DIS
LIN {X 64.2437,Y -43.3173,Z 80,A -39.7937,B 24.9104,C -2.1853,E1 25.1316,E2 124.4036} C_DIS
LIN {X 61.4745,Y -47.1649,Z 80,A -43.4287,B 24.9115,C -2.172,E1 25.1256,E2 128.0528} C_DIS
LIN {X 59.493,Y -49.6411,Z 80,A -45.6162,B 24.9116,C -2.1706,E1 25.1217,E2 130.2333} C_DIS
LIN {X 57.2704,Y -52.1901,Z 80,A -48.0362,B 24.9119,C -2.1667,E1 25.1172,E2 132.6517} C_DIS
LIN {X 54.5779,Y -54.9992,Z 80,A -51.0866,B 24.9129,C -2.1545,E1 25.1112,E2 135.7179} C_DIS
LIN {X 52.0804,Y -57.3702,Z 80,A -53.4747,B 24.913,C -2.1533,E1 25.1064,E2 138.0991} C_DIS
LIN {X 49.5589,Y -59.5612,Z 80,A -55.9503,B 24.9135,C -2.1477,E1 25.1011,E2 140.5785} C_DIS
LIN {X 46.3134,Y -62.119,Z 80,A -59.3795,B 24.9149,C -2.1301,E1 25.0934,E2 144.0367} C_DIS
LIN {X 42.6376,Y -64.6967,Z 80,A -62.3057,B 24.9145,C -2.1352,E1 25.0867,E2 146.941} C_DIS
LIN {X 39.8565,Y -66.4473,Z 80,A -64.7186,B 24.9148,C -2.1311,E1 25.081,E2 149.3559} C_DIS
LIN {X 36.4531,Y -68.3732,Z 80,A -68.35,B 24.9169,C -2.1046,E1 25.0719,E2 153.0396} C_DIS
LIN {X 33.005,Y -70.1026,Z 80,A -70.4132,B 24.9155,C -2.123,E1 25.0669,E2 155.054} C_DIS
LIN {X 29.5225,Y -71.6381,Z 80,A -73.3684,B 24.9161,C -2.1148,E1 25.0593,E2 158.0215} C_DIS
LIN {X 26.0214,Y -72.9825,Z 80,A -75.5594,B 24.9151,C -2.128,E1 25.0536,E2 160.1765} C_DIS
LIN {X 21.5984,Y -74.4133,Z 80,A -79.5484,B 24.9167,C -2.108,E1 25.0429,E2 164.2056} C_DIS
LIN {X 17.9732,Y -75.3693,Z 80,A -82.1421,B 24.9165,C -2.1103,E1 25.0359,E2 166.7899} C_DIS
LIN {X 12.0971,Y -76.5334,Z 80,A -86.5208,B 24.9167,C -2.1081,E1 25.0239,E2 171.1687} C_DIS
LIN {X 6.9807,Y -77.1681,Z 80,A -90.0093,B 24.9161,C -2.115,E1 25.0143,E2 174.6384} C_DIS
LIN {X 4.4449,Y -77.3557,Z 80,A -92.1899,B 24.9168,C -2.1057,E1 25.0081,E2 176.8401} C_DIS
LIN {X 1.144,Y -77.4744,Z 80,A -94.7392,B 24.9171,C -2.102,E1 25.001,E2 179.3977} C_DIS
LIN {X 1.144,Y -77.4744,Z 80,A -94.7392,B 24.9171,C -2.102,E1 25.001,E2 179.3977} C_DIS
Enddeposition()
LIN {X 0.483,Y -76.5778,Z 80,A -94.1824,B 24.9136,C -2.1467,E1 25.0028,E2 178.7347} C_DIS
Startdeposition()
$VEL.CP = VEL_PRINT
LIN {X 4.1909,Y -76.4741,Z 80,A -91.5055,B 24.9137,C -2.1448,E1 25.0103,E2 176.0632} C_DIS
LIN {X 6.8147,Y -76.2856,Z 80,A -89.1226,B 24.9127,C -2.1575,E1 25.017,E2 173.6513} C_DIS
LIN {X 11.0499,Y -75.7881,Z 80,A -86.4529,B 24.9137,C -2.1447,E1 25.0243,E2 171.0141} C_DIS
LIN {X 13.4038,Y -75.407,Z 80,A -83.9874,B 24.912,C -2.1656,E1 25.0312,E2 168.5017} C_DIS
LIN {X 18.2061,Y -74.3937,Z 80,A -80.7244,B 24.9127,C -2.1572,E1 25.04,E2 165.263} C_DIS
LIN {X 21.1471,Y -73.6121,Z 80,A -77.2092,B 24.9095,C -2.196,E1 25.0497,E2 161.662} C_DIS
LIN {X 26.1294,Y -71.994,Z 80,A -74.8797,B 24.913,C -2.1543,E1 25.0556,E2 159.436} C_DIS
LIN {X 28.0625,Y -71.2627,Z 80,A -72.1843,B 24.91,C -2.1901,E1 25.0628,E2 156.6617} C_DIS
LIN {X 31.7807,Y -69.6841,Z 80,A -70.2383,B 24.9123,C -2.1629,E1 25.0676,E2 154.7849} C_DIS
LIN {X 35.0216,Y -68.1131,Z 80,A -67.3836,B 24.9115,C -2.172,E1 25.0747,E2 151.9164} C_DIS
LIN {X 39.1619,Y -65.82,Z 80,A -63.8044,B 24.9109,C -2.1794,E1 25.0834,E2 148.3303} C_DIS
LIN {X 41.8982,Y -64.1132,Z 80,A -61.5433,B 24.9109,C -2.1794,E1 25.0887,E2 146.0764} C_DIS
LIN {X 45.7235,Y -61.444,Z 80,A -57.5063,B 24.909,C -2.2029,E1 25.098,E2 141.9979} C_DIS
LIN {X 49.1699,Y -58.722,Z 80,A -54.6394,B 24.9094,C -2.1975,E1 25.1042,E2 139.1547} C_DIS
LIN {X 51.9815,Y -56.2483,Z 80,A -51.4751,B 24.908,C -2.2149,E1 25.1108,E2 135.962} C_DIS
LIN {X 56.0395,Y -52.207,Z 80,A -47.5552,B 24.908,C -2.2143,E1 25.1184,E2 132.0604} C_DIS
LIN {X 58.2277,Y -49.7536,Z 80,A -45.2619,B 24.908,C -2.2155,E1 25.1226,E2 129.7746} C_DIS
LIN {X 60.8995,Y -46.4459,Z 80,A -41.8405,B 24.9066,C -2.2312,E1 25.1285,E2 126.3321} C_DIS
LIN {X 63.2704,Y -43.1601,Z 80,A -38.9855,B 24.9064,C -2.2341,E1 25.1331,E2 123.4843} C_DIS
LIN {X 64.8151,Y -40.8039,Z 80,A -35.9783,B 24.9035,C -2.2678,E1 25.1377,E2 120.4126} C_DIS
LIN {X 66.9708,Y -37.1595,Z 80,A -33.8321,B 24.9054,C -2.2453,E1 25.1405,E2 118.3306} C_DIS
LIN {X 68.9579,Y -33.3266,Z 80,A -30.5283,B 24.9044,C -2.2571,E1 25.1447,E2 115.0166} C_DIS
LIN {X 71.365,Y -27.8014,Z 80,A -26.2365,B 24.9038,C -2.264,E1 25.1494,E2 110.7321} C_DIS
LIN {X 73.3379,Y -22.0772,Z 80,A -21.5946,B 24.9024,C -2.2814,E1 25.1535,E2 106.0754} C_DIS
LIN {X 74.172,Y -19.089,Z 80,A -19.0939,B 24.9013,C -2.2942,E1 25.1553,E2 103.5587} C_DIS
LIN {X 74.8363,Y -16.2909,Z 80,A -16.3963,B 24.8992,C -2.318,E1 25.1569,E2 100.8207} C_DIS
LIN {X 75.5326,Y -12.6767,Z 80,A -14.9072,B 24.9018,C -2.2875,E1 25.1576,E2 99.4123} C_DIS
LIN {X 76.0592,Y -8.9893,Z 80,A -11.8196,B 24.9003,C -2.3056,E1 25.1588,E2 96.3001} C_DIS
LIN {X 76.3178,Y -6.4445,Z 80,A -9.6647,B 24.8991,C -2.3191,E1 25.1594,E2 94.126} C_DIS
LIN {X 76.5209,Y -3.2301,Z 80,A -7.6794,B 24.8996,C -2.3137,E1 25.1597,E2 92.1652} C_DIS
LIN {X 76.5873,Y 0.4864,Z 80,A -3.8069,B 24.8958,C -2.3565,E1 25.1597,E2 88.2149} C_DIS
LIN {X 76.47,Y 4.268,Z 80,A -1.7262,B 24.8971,C -2.3421,E1 25.1594,E2 86.1805} C_DIS
LIN {X 76.2983,Y 6.6772,Z 80,A 0.2575,B 24.8961,C -2.3532,E1 25.159,E2 84.1823} C_DIS
LIN {X 75.8156,Y 10.8572,Z 80,A 3.2335,B 24.8957,C -2.3578,E1 25.1579,E2 81.213} C_DIS
LIN {X 75.3762,Y 13.5757,Z 80,A 5.3921,B 24.8948,C -2.3672,E1 25.1568,E2 79.0448} C_DIS
LIN {X 74.403,Y 18.1679,Z 80,A 8.7272,B 24.8944,C -2.3725,E1 25.1548,E2 75.7166} C_DIS
LIN {X 73.5275,Y 21.4408,Z 80,A 10.9519,B 24.8945,C -2.3706,E1 25.1532,E2 73.5091} C_DIS
LIN {X 72.2381,Y 25.447,Z 80,A 14.4047,B 24.8929,C -2.3892,E1 25.1501,E2 70.0319} C_DIS
LIN {X 70.4752,Y 29.9858,Z 80,A 17.9869,B 24.8921,C -2.3978,E1 25.1464,E2 66.4492} C_DIS
LIN {X 69.6097,Y 31.9423,Z 80,A 19.8018,B 24.8911,C -2.4089,E1 25.1443,E2 64.618} C_DIS
LIN {X 67.9093,Y 35.4143,Z 80,A 22.4087,B 24.8911,C -2.4081,E1 25.141,E2 62.0268} C_DIS
LIN {X 65.4749,Y 39.7356,Z 80,A 26.7511,B 24.8885,C -2.4371,E1 25.1348,E2 57.6382} C_DIS
LIN {X 63.6246,Y 42.637,Z 80,A 28.6447,B 24.8898,C -2.423,E1 25.1319,E2 55.7873} C_DIS
LIN {X 61.2751,Y 45.9483,Z 80,A 32.1449,B 24.8879,C -2.4444,E1 25.1261,E2 52.2535} C_DIS
LIN {X 58.5924,Y 49.3253,Z 80,A 35.6794,B 24.8863,C -2.4611,E1 25.1198,E2 48.6957} C_DIS
LIN {X 56.0794,Y 52.1647,Z 80,A 38.5157,B 24.8857,C -2.4673,E1 25.1144,E2 45.8572} C_DIS
LIN {X 53.4088,Y 54.8954,Z 80,A 40.6129,B 24.8873,C -2.4506,E1 25.1103,E2 43.8083} C_DIS
LIN {X 50.777,Y 57.338,Z 80,A 43.3068,B 24.8868,C -2.4562,E1 25.1047,E2 41.112} C_DIS
LIN {X 47.8942,Y 59.7679,Z 80,A 46.1018,B 24.8864,C -2.4607,E1 25.0987,E2 38.3171} C_DIS
LIN {X 44.5457,Y 62.3022,Z 80,A 49.736,B 24.8845,C -2.4805,E1 25.0904,E2 34.6487} C_DIS
LIN {X 41.3502,Y 64.4674,Z 80,A 52.8666,B 24.8834,C -2.4921,E1 25.0831,E2 31.5009} C_DIS
LIN {X 38.0345,Y 66.4776,Z 80,A 55.1908,B 24.8846,C -2.4794,E1 25.0775,E2 29.2137} C_DIS
LIN {X 35.1453,Y 68.0499,Z 80,A 57.7047,B 24.8842,C -2.4842,E1 25.0713,E2 26.6957} C_DIS
LIN {X 30.4272,Y 70.2848,Z 80,A 61.3434,B 24.8845,C -2.481,E1 25.0621,E2 23.0737} C_DIS
LIN {X 27.4187,Y 71.5135,Z 80,A 64.2623,B 24.8829,C -2.4972,E1 25.0544,E2 20.1227} C_DIS
LIN {X 23.758,Y 72.8111,Z 80,A 67.3179,B 24.8823,C -2.5038,E1 25.0463,E2 17.0572} C_DIS
LIN {X 20.3969,Y 73.8226,Z 80,A 69.1235,B 24.8843,C -2.4825,E1 25.0416,E2 15.3053} C_DIS
LIN {X 17.5801,Y 74.5442,Z 80,A 71.0919,B 24.8847,C -2.478,E1 25.0363,E2 13.3505} C_DIS
LIN {X 14.2062,Y 75.2604,Z 80,A 74.3224,B 24.883,C -2.4972,E1 25.0273,E2 10.0784} C_DIS
LIN {X 10.9756,Y 75.7988,Z 80,A 76.6611,B 24.8832,C -2.4947,E1 25.0209,E2 7.7476} C_DIS
LIN {X 7.1075,Y 76.2585,Z 80,A 79.4102,B 24.8836,C -2.4906,E1 25.0133,E2 5.0102} C_DIS
LIN {X 2.8224,Y 76.5366,Z 80,A 82.5841,B 24.8836,C -2.4895,E1 25.0044,E2 1.8401} C_DIS
LIN {X -0.4727,Y 76.5876,Z 80,A 84.96,B 24.8839,C -2.4866,E1 24.9978,E2 -0.5288} C_DIS
LIN {X -5.3491,Y 76.4022,Z 80,A 88.6785,B 24.8839,C -2.4871,E1 24.9875,E2 -4.2495} C_DIS
Enddeposition()
END
